C01811=1012.255,117.032,374.346,169.499,79.664,168.490
C01812=1012.256,116.639,374.386,169.507,79.676,168.501
C01813=1012.257,116.245,374.424,169.516,79.687,168.512
C01814=1012.259,115.850,374.464,169.527,79.699,168.525
C01815=1012.260,115.456,374.502,169.537,79.712,168.537
C01816=1012.261,115.062,374.541,169.547,79.725,168.549
C01817=1012.262,114.667,374.580,169.559,79.737,168.563
C01818=1012.263,114.273,374.619,169.567,79.748,168.573
C01819=1012.264,113.879,374.658,169.578,79.759,168.585
C01820=1012.266,113.484,374.697,169.586,79.770,168.596
C01821=1012.267,113.090,374.735,169.596,79.781,168.607
C01822=1012.269,112.696,374.774,169.607,79.793,168.620
C01823=1012.270,112.302,374.813,169.618,79.805,168.633
C01824=1012.271,111.908,374.852,169.629,79.818,168.646
C01825=1012.272,111.514,374.890,169.637,79.830,168.657
C01826=1012.273,111.119,374.929,169.651,79.841,168.671
C01827=1012.274,110.725,374.968,169.660,79.852,168.682
C01828=1012.275,110.331,375.007,169.670,79.863,168.694
C01829=1012.277,109.936,375.046,169.677,79.873,168.704
C01830=1012.278,109.542,375.084,169.689,79.885,168.717
C01831=1012.280,109.148,375.123,169.700,79.898,168.730
C01832=1012.280,108.754,375.162,169.709,79.909,168.741
C01833=1012.282,108.359,375.200,169.721,79.921,168.755
C01834=1012.283,107.965,375.239,169.730,79.932,168.766
C01835=1012.284,107.570,375.278,169.740,79.943,168.778
C01836=1012.285,107.176,375.316,169.751,79.954,168.790
C01837=1012.286,106.782,375.355,169.761,79.964,168.802
C01838=1012.287,106.388,375.394,169.771,79.976,168.814
C01839=1012.289,105.993,375.431,169.780,79.987,168.825
C01840=1012.290,105.599,375.470,169.792,79.999,168.839
C01841=1012.291,105.205,375.509,169.801,80.010,168.850
C01842=1012.292,104.811,375.547,169.815,80.022,168.865
C01843=1012.293,104.416,375.585,169.825,80.033,168.877
C01844=1012.295,104.022,375.624,169.832,80.043,168.886
C01845=1012.296,103.628,375.663,169.845,80.053,168.899
C01846=1012.296,103.233,375.702,169.852,80.063,168.909
C01847=1012.298,102.838,375.740,169.865,80.075,168.923
C01848=1012.299,102.444,375.778,169.877,80.087,168.937
C01849=1012.300,102.049,375.816,169.887,80.098,168.949
C01850=1012.301,101.655,375.855,169.898,80.109,168.962
C01851=1012.302,101.261,375.893,169.909,80.120,168.974
C01852=1012.304,100.866,375.932,169.920,80.130,168.987
C01853=1012.305,100.472,375.970,169.928,80.140,168.996
C01854=1012.307,100.077,376.008,169.937,80.149,169.007
C01855=1012.307,99.683,376.046,169.950,80.161,169.022
C01856=1012.309,99.288,376.085,169.960,80.173,169.033
C01857=1012.310,98.894,376.124,169.973,80.185,169.048
C01858=1012.311,98.499,376.161,169.984,80.196,169.061
C01859=1012.312,98.105,376.200,169.995,80.206,169.073
C01860=1012.313,97.710,376.238,170.003,80.216,169.083
C01861=1012.314,97.316,376.276,170.016,80.226,169.097
C01862=1012.316,96.921,376.314,170.025,80.235,169.108
C01863=1012.317,96.527,376.353,170.037,80.246,169.121
C01864=1012.318,96.133,376.391,170.047,80.257,169.133
C01865=1012.319,95.737,376.429,170.057,80.269,169.145
C01866=1012.320,95.343,376.467,170.068,80.279,169.158
C01867=1012.321,94.949,376.505,170.080,80.290,169.171
C01868=1012.322,94.554,376.543,170.089,80.299,169.182
C01869=1012.323,94.160,376.581,170.101,80.310,169.195
C01870=1012.325,93.765,376.619,170.111,80.319,169.206
C01871=1012.326,93.370,376.658,170.120,80.328,169.217
C01872=1012.327,92.976,376.696,170.132,80.339,169.230
C01873=1012.328,92.581,376.734,170.140,80.349,169.240
C01874=1012.329,92.186,376.772,170.152,80.360,169.253
C01875=1012.331,91.792,376.810,170.164,80.370,169.267
C01876=1012.332,91.397,376.847,170.176,80.381,169.280
C01877=1012.332,90.994,376.887,170.188,80.391,169.293
C01878=1012.333,90.749,376.911,170.195,80.397,169.301
C01879=1012.334,90.468,376.937,170.200,80.404,169.308
C01880=1012.335,90.194,376.963,170.207,80.410,169.316
C01881=1012.335,89.959,376.986,170.214,80.416,169.323
C01882=1012.336,89.564,377.024,170.224,80.426,169.334
C01883=1012.338,89.178,377.061,170.237,80.436,169.348
C01884=1012.339,88.800,377.097,170.246,80.445,169.359
C01885=1012.340,88.425,377.133,170.256,80.455,169.370
C01886=1012.341,88.047,377.170,170.266,80.464,169.382
C01887=1012.342,87.663,377.207,170.279,80.474,169.396
C01888=1012.343,87.269,377.244,170.288,80.484,169.407
C01889=1012.344,86.870,377.282,170.298,80.493,169.418
C01890=1012.345,86.469,377.320,170.311,80.504,169.432
C01891=1012.346,86.067,377.359,170.321,80.513,169.443
C01892=1012.347,85.664,377.398,170.333,80.524,169.457
C01893=1012.349,85.260,377.437,170.343,80.533,169.469
C01894=1012.350,84.853,377.476,170.356,80.543,169.482
C01895=1012.351,84.447,377.514,170.366,80.553,169.494
C01896=1012.352,84.039,377.554,170.378,80.563,169.508
C01897=1012.352,83.629,377.592,170.389,80.573,169.520
C01898=1012.354,83.218,377.632,170.401,80.583,169.533
C01899=1012.355,82.805,377.671,170.412,80.592,169.545
C01900=1012.356,82.393,377.710,170.424,80.603,169.559
C01901=1012.357,81.979,377.750,170.435,80.612,169.571
C01902=1012.358,81.565,377.789,170.447,80.623,169.585
C01903=1012.360,81.171,377.827,170.458,80.632,169.597
C01904=1012.360,80.807,377.862,170.470,80.641,169.609
C01905=1012.362,80.424,377.898,170.481,80.650,169.621
C01906=1012.363,80.012,377.936,170.490,80.660,169.633
C01907=1012.363,79.603,377.976,170.501,80.669,169.645
C01908=1012.364,79.201,378.014,170.511,80.678,169.657
C01909=1012.366,78.806,378.051,170.526,80.688,169.672
C01910=1012.366,78.417,378.088,170.536,80.698,169.684
C01911=1012.368,78.033,378.125,170.545,80.705,169.694
C01912=1012.368,77.652,378.161,170.556,80.715,169.706
C01913=1012.370,77.270,378.197,170.567,80.724,169.718
C01914=1012.371,76.884,378.234,170.578,80.733,169.730
C01915=1012.371,76.489,378.271,170.590,80.742,169.743
C01916=1012.372,76.088,378.309,170.601,80.751,169.755
C01917=1012.373,75.678,378.347,170.612,80.760,169.767
C01918=1012.374,75.264,378.387,170.623,80.769,169.780
C01919=1012.375,75.055,378.407,170.628,80.774,169.786
C01920=1012.376,74.840,378.427,170.636,80.780,169.794
C01921=1012.376,74.614,378.448,170.642,80.784,169.801
C01922=1012.377,74.385,378.470,170.647,80.789,169.807
C01923=1012.378,74.166,378.490,170.656,80.795,169.815
C01924=1012.379,73.752,378.530,170.667,80.804,169.828
C01925=1012.380,73.339,378.569,170.678,80.813,169.840
C01926=1012.381,72.930,378.607,170.689,80.823,169.853
C01927=1012.382,72.522,378.645,170.700,80.832,169.865
C01928=1012.383,72.116,378.683,170.711,80.841,169.878
C01929=1012.384,71.711,378.722,170.724,80.850,169.891
C01930=1012.384,71.306,378.760,170.735,80.859,169.903
C01931=1012.385,70.901,378.798,170.747,80.868,169.916
C01932=1012.386,70.497,378.836,170.756,80.876,169.926
C01933=1012.387,70.093,378.874,170.767,80.885,169.939
C01934=1012.388,69.689,378.912,170.779,80.894,169.952
C01935=1012.390,69.280,378.951,170.792,80.903,169.965
C01936=1012.391,68.864,378.989,170.803,80.912,169.978
C01937=1012.392,68.447,379.029,170.815,80.921,169.991
C01938=1012.393,68.035,379.067,170.824,80.929,170.001
C01939=1012.393,67.634,379.105,170.835,80.938,170.014
C01940=1012.395,67.235,379.142,170.848,80.947,170.027
C01941=1012.395,66.838,379.179,170.856,80.956,170.037
C01942=1012.396,66.474,379.213,170.867,80.963,170.049
C01943=1012.397,66.147,379.243,170.877,80.970,170.059
C01944=1012.398,65.754,379.281,170.886,80.978,170.070
C01945=1012.398,65.546,379.300,170.893,80.983,170.077
C01946=1012.399,65.331,379.320,170.899,80.987,170.084
C01947=1012.400,65.112,379.340,170.905,80.992,170.090
C01948=1012.400,64.890,379.361,170.911,80.996,170.097
C01949=1012.401,64.663,379.382,170.920,81.002,170.106
C01950=1012.401,64.436,379.403,170.926,81.006,170.113
C01951=1012.402,64.217,379.424,170.932,81.011,170.119
C01952=1012.402,63.813,379.460,170.977,81.046,170.169
C01953=1012.402,63.601,379.477,171.070,81.117,170.271
C01954=1012.402,63.366,379.495,171.175,81.195,170.386
C01955=1012.402,63.117,379.514,171.288,81.278,170.511
C01956=1012.402,62.875,379.533,171.401,81.358,170.633
C01957=1012.402,62.656,379.550,171.504,81.430,170.745
C01958=1012.402,62.372,379.572,171.641,81.524,170.894
C01959=1012.402,61.974,379.603,171.838,81.655,171.108
C01960=1012.402,61.578,379.633,172.039,81.784,171.326
C01961=1012.403,61.182,379.664,172.249,81.914,171.552
C01962=1012.402,60.785,379.695,172.466,82.043,171.786
C01963=1012.403,60.389,379.726,172.690,82.171,172.025
C01964=1012.403,59.993,379.756,172.921,82.299,172.272
C01965=1012.402,59.598,379.787,173.157,82.427,172.524
C01966=1012.403,59.201,379.818,173.408,82.554,172.791
C01967=1012.403,58.805,379.848,173.660,82.680,173.059
C01968=1012.403,58.409,379.880,173.927,82.807,173.341
C01969=1012.403,58.013,379.910,174.202,82.932,173.630
C01970=1012.403,57.616,379.940,174.486,83.058,173.930
C01971=1012.403,57.221,379.972,174.784,83.183,174.242
C01972=1012.403,56.824,380.002,175.090,83.306,174.562
C01973=1012.404,56.429,380.033,175.408,83.430,174.895
C01974=1012.404,56.033,380.063,175.735,83.552,175.237
C01975=1012.404,55.636,380.094,176.082,83.675,175.597
C01976=1012.404,55.241,380.125,176.433,83.797,175.963
C01977=1012.404,54.844,380.155,176.806,83.918,176.349
C01978=1012.405,54.448,380.186,177.189,84.039,176.746
C01979=1012.404,54.052,380.217,177.590,84.158,177.160
C01980=1012.405,53.656,380.247,178.004,84.277,177.588
C01981=1012.405,53.260,380.278,178.436,84.396,178.033
C01982=1012.406,52.865,380.309,178.889,84.513,178.499
C01983=1012.406,52.469,380.339,179.364,84.631,178.987
C01984=1012.407,52.072,380.370,179.855,84.746,179.490
C01985=1012.407,51.677,380.400,-179.631,84.863,-179.983
C01986=1012.407,51.281,380.431,-179.099,84.977,-179.438
C01987=1012.407,50.884,380.461,-178.540,85.091,-178.867
C01988=1012.407,50.489,380.492,-177.953,85.203,-178.268
C01989=1012.408,50.093,380.522,-177.344,85.315,-177.647
C01990=1012.408,49.697,380.553,-176.695,85.427,-176.986
C01991=1012.409,49.301,380.584,-176.030,85.537,-176.309
C01992=1012.409,48.905,380.614,-175.320,85.647,-175.588
C01993=1012.410,48.508,380.645,-174.582,85.754,-174.838
C01994=1012.410,48.114,380.675,-173.803,85.862,-174.048
C01995=1012.411,47.717,380.706,-172.982,85.967,-173.216
C01996=1012.411,47.321,380.736,-172.125,86.072,-172.348
C01997=1012.412,46.926,380.767,-171.221,86.176,-171.432
C01998=1012.412,46.530,380.798,-170.277,86.277,-170.478
C01999=1012.411,46.134,380.828,-169.265,86.378,-169.456
C02000=1012.413,45.739,380.859,-168.208,86.477,-168.388
C02001=1012.413,45.342,380.889,-167.101,86.574,-167.271
C02002=1012.413,44.947,380.920,-165.914,86.670,-166.074
C02003=1012.414,44.551,380.950,-164.672,86.764,-164.822
C02004=1012.414,44.155,380.982,-163.370,86.855,-163.509
C02005=1012.415,43.760,381.011,-161.972,86.945,-162.102
C02006=1012.415,43.364,381.042,-160.504,87.033,-160.624
C02007=1012.416,42.969,381.073,-158.950,87.118,-159.060
C02008=1012.416,42.572,381.103,-157.318,87.201,-157.418
C02009=1012.417,42.177,381.134,-155.591,87.280,-155.683
C02010=1012.417,41.781,381.165,-153.754,87.358,-153.836
C02011=1012.418,41.386,381.194,-151.813,87.432,-151.886
C02012=1012.418,40.990,381.225,-149.777,87.502,-149.842
C02013=1012.419,40.594,381.256,-147.632,87.569,-147.689
C02014=1012.419,40.200,381.286,-145.391,87.631,-145.438
C02015=1012.420,39.803,381.317,-143.005,87.690,-143.044
C02016=1012.420,39.408,381.347,-140.520,87.745,-140.550
C02017=1012.421,39.012,381.378,-137.951,87.794,-137.973
C02018=1012.422,38.616,381.408,-135.243,87.839,-135.257
C02019=1012.423,38.221,381.439,-132.449,87.879,-132.455
C02020=1012.423,37.825,381.469,-129.568,87.913,-129.567
C02021=1012.423,37.430,381.499,-126.623,87.942,-126.613
C02022=1012.424,37.035,381.530,-123.575,87.965,-123.558
C02023=1012.424,36.639,381.561,-120.534,87.982,-120.509
C02024=1012.425,36.243,381.591,-117.404,87.993,-117.372
C02025=1012.426,35.849,381.622,-114.310,87.998,-114.271
C02026=1012.427,35.453,381.652,-111.189,87.997,-111.142
C02027=1012.427,35.057,381.682,-108.098,87.990,-108.044
C02028=1012.428,34.662,381.713,-105.036,87.977,-104.976
C02029=1012.429,34.266,381.743,-102.042,87.959,-101.975
C02030=1012.430,33.871,381.774,-99.149,87.936,-99.074
C02031=1012.430,33.475,381.804,-96.307,87.906,-96.226
C02032=1012.430,33.080,381.835,-93.566,87.873,-93.479
C02033=1012.431,32.685,381.865,-90.937,87.834,-90.843
C02034=1012.432,32.290,381.896,-88.403,87.792,-88.303
C02035=1012.433,31.894,381.926,-85.985,87.745,-85.878
C02036=1012.433,31.499,381.957,-83.686,87.695,-83.574
C02037=1012.434,31.103,381.987,-81.471,87.641,-81.352
C02038=1012.434,30.708,382.018,-79.404,87.585,-79.280
C02039=1012.435,30.313,382.047,-77.406,87.524,-77.277
C02040=1012.436,29.917,382.078,-75.542,87.463,-75.406
C02041=1012.436,29.522,382.108,-73.759,87.398,-73.618
C02042=1012.437,29.127,382.139,-72.088,87.331,-71.941
C02043=1012.438,28.732,382.169,-70.499,87.263,-70.348
C02044=1012.439,28.338,382.200,-68.990,87.192,-68.833
C02045=1012.439,27.944,382.230,-67.576,87.120,-67.414
C02046=1012.440,27.552,382.260,-66.231,87.047,-66.065
C02047=1012.441,27.158,382.291,-64.958,86.973,-64.786
C02048=1012.441,26.764,382.321,-63.759,86.898,-63.582
C02049=1012.442,26.368,382.352,-62.613,86.821,-62.432
C02050=1012.443,25.970,382.383,-61.514,86.743,-61.328
C02051=1012.443,25.570,382.413,-60.479,86.664,-60.288
C02052=1012.444,25.174,382.443,-59.503,86.584,-59.308
C02053=1012.445,24.779,382.474,-58.575,86.504,-58.376
C02054=1012.446,24.383,382.504,-57.689,86.424,-57.485
C02055=1012.447,24.004,382.534,-56.888,86.347,-56.681
C02056=1012.447,23.664,382.560,-56.198,86.277,-55.987
C02057=1012.448,23.248,382.591,-55.397,86.192,-55.182
C02058=1012.448,22.884,382.620,-54.721,86.116,-54.503
C02059=1012.449,22.606,382.641,-54.231,86.059,-54.009
C02060=1012.450,22.275,382.667,-53.666,85.990,-53.442
C02061=1012.450,21.947,382.692,-53.123,85.921,-52.895
C02062=1012.451,21.558,382.721,-52.509,85.841,-52.278
C02063=1012.451,21.330,382.740,-52.158,85.793,-51.925
C02064=1012.452,21.083,382.759,-51.791,85.742,-51.556
C02065=1012.452,20.822,382.778,-51.416,85.687,-51.178
C02066=1012.453,20.554,382.799,-51.042,85.631,-50.802
C02067=1012.454,20.285,382.819,-50.678,85.576,-50.436
C02068=1012.454,20.024,382.840,-50.331,85.521,-50.087
C02069=1012.455,19.782,382.858,-50.022,85.471,-49.776
C02070=1012.455,19.561,382.875,-49.742,85.424,-49.494
C02071=1012.456,19.358,382.891,-49.496,85.383,-49.247
C02072=1012.456,18.955,382.922,-49.018,85.299,-48.766
C02073=1012.457,18.555,382.952,-48.564,85.216,-48.309
C02074=1012.457,18.163,382.983,-48.132,85.135,-47.873
C02075=1012.458,17.773,383.013,-47.720,85.053,-47.459
C02076=1012.460,17.386,383.043,-47.329,84.973,-47.065
C02077=1012.460,16.999,383.073,-46.955,84.894,-46.689
C02078=1012.460,16.615,383.102,-46.594,84.815,-46.325
C02079=1012.461,16.232,383.131,-46.249,84.737,-45.978
C02080=1012.462,15.851,383.161,-45.914,84.658,-45.641
C02081=1012.463,15.471,383.190,-45.594,84.581,-45.319
C02082=1012.464,15.090,383.220,-45.284,84.503,-45.006
C02083=1012.464,14.710,383.249,-44.988,84.426,-44.709
C02084=1012.465,14.330,383.278,-44.699,84.350,-44.418
C02085=1012.466,13.949,383.307,-44.419,84.273,-44.136
C02086=1012.467,13.567,383.337,-44.146,84.196,-43.861
C02087=1012.468,13.184,383.366,-43.885,84.121,-43.598
C02088=1012.468,12.800,383.396,-43.626,84.044,-43.337
C02089=1012.468,12.416,383.425,-43.379,83.967,-43.089
C02090=1012.470,12.034,383.454,-43.142,83.892,-42.851
C02091=1012.470,11.662,383.483,-42.919,83.820,-42.626
C02092=1012.471,11.298,383.511,-42.705,83.749,-42.409
C02093=1012.472,10.933,383.540,-42.496,83.677,-42.200
C02094=1012.472,10.559,383.568,-42.292,83.605,-41.995
C02095=1012.473,10.181,383.598,-42.089,83.533,-41.790
C02096=1012.474,9.805,383.626,-41.894,83.461,-41.594
C02097=1012.475,9.431,383.655,-41.703,83.390,-41.401
C02098=1012.475,9.057,383.684,-41.520,83.319,-41.218
C02099=1012.475,8.683,383.713,-41.342,83.248,-41.038
C02100=1012.477,8.309,383.741,-41.166,83.178,-40.861
C02101=1012.478,7.933,383.771,-40.998,83.108,-40.692
C02102=1012.478,7.555,383.799,-40.833,83.039,-40.527
C02103=1012.479,7.173,383.828,-40.668,82.968,-40.361
C02104=1012.480,6.788,383.858,-40.512,82.898,-40.204
C02105=1012.480,6.396,383.888,-40.353,82.827,-40.045
C02106=1012.482,6.004,383.919,-40.199,82.755,-39.890
C02107=1012.481,5.611,383.949,-40.051,82.685,-39.742
C02108=1012.483,5.220,383.979,-39.906,82.615,-39.596
C02109=1012.483,4.832,384.009,-39.766,82.546,-39.455
C02110=1012.485,4.442,384.039,-39.628,82.478,-39.317
C02111=1012.485,4.051,384.070,-39.493,82.410,-39.180
C02112=1012.486,3.679,384.098,-39.371,82.345,-39.060
C02113=1012.487,3.335,384.125,-39.259,82.285,-38.947
C02114=1012.487,3.010,384.149,-39.155,82.230,-38.843
C02115=1012.487,2.687,384.174,-39.056,82.175,-38.743
C02116=1012.489,2.345,384.201,-38.951,82.117,-38.638
C02117=1012.488,1.974,384.229,-38.840,82.055,-38.527
C02118=1012.490,1.582,384.260,-38.727,81.989,-38.414
C02119=1012.490,1.185,384.290,-38.616,81.924,-38.303
C02120=1012.491,0.788,384.321,-38.507,81.858,-38.194
C02121=1012.492,0.394,384.351,-38.402,81.794,-38.089
C02122=1012.492,-0.001,384.381,-38.298,81.730,-37.985
C02123=1012.493,-0.399,384.412,-38.196,81.666,-37.883
C02124=1012.494,-0.800,384.443,-38.099,81.602,-37.787
C02125=1012.494,-1.202,384.474,-37.999,81.539,-37.686
C02126=1012.496,-1.606,384.505,-37.905,81.475,-37.593
C02127=1012.496,-2.013,384.536,-37.811,81.413,-37.499
C02128=1012.497,-2.422,384.568,-37.719,81.350,-37.407
C02129=1012.497,-2.832,384.599,-37.630,81.288,-37.319
C02130=1012.498,-3.244,384.631,-37.543,81.226,-37.233
C02131=1012.498,-3.645,384.662,-37.458,81.166,-37.148
C02132=1012.499,-4.031,384.691,-37.381,81.109,-37.071
C02133=1012.500,-4.410,384.721,-37.307,81.053,-36.998
C02134=1012.501,-4.801,384.751,-37.229,80.996,-36.920
C02135=1012.501,-5.215,384.783,-37.151,80.937,-36.843
C02136=1012.502,-5.430,384.800,-37.110,80.906,-36.802
C02137=1012.501,-5.646,384.816,-37.074,80.875,-36.767
C02138=1012.502,-5.863,384.833,-37.034,80.844,-36.727
C02139=1012.503,-6.080,384.850,-36.994,80.813,-36.687
C02140=1012.503,-6.296,384.866,-36.957,80.783,-36.651
C02141=1012.504,-6.513,384.883,-36.919,80.754,-36.613
C02142=1012.504,-6.729,384.899,-36.883,80.724,-36.578
C02143=1012.505,-6.945,384.917,-36.845,80.695,-36.540
C02144=1012.505,-7.159,384.933,-36.809,80.664,-36.505
C02145=1012.504,-7.374,384.949,-36.775,80.636,-36.471
C02146=1012.506,-7.587,384.966,-36.739,80.607,-36.435
C02147=1012.505,-7.800,384.983,-36.705,80.578,-36.401
C02148=1012.506,-8.013,384.999,-36.671,80.549,-36.368
C02149=1012.506,-8.224,385.015,-36.639,80.522,-36.337
C02150=1012.506,-8.436,385.032,-36.606,80.494,-36.304
C02151=1012.506,-8.647,385.048,-36.574,80.467,-36.273
C02152=1012.507,-8.858,385.064,-36.541,80.438,-36.241
C02153=1012.508,-9.070,385.081,-36.510,80.411,-36.210
C02154=1012.508,-9.281,385.097,-36.479,80.384,-36.179
C02155=1012.508,-9.703,385.129,-36.419,80.330,-36.121
C02156=1012.509,-10.124,385.162,-36.360,80.278,-36.062
C02157=1012.509,-10.544,385.194,-36.302,80.224,-36.006
C02158=1012.511,-10.963,385.226,-36.245,80.173,-35.949
C02159=1012.511,-11.381,385.259,-36.191,80.123,-35.896
C02160=1012.512,-11.797,385.291,-36.137,80.072,-35.843
C02161=1012.512,-12.212,385.322,-36.085,80.024,-35.792
C02162=1012.513,-12.625,385.354,-36.036,79.975,-35.745
C02163=1012.514,-13.034,385.386,-35.986,79.928,-35.696
C02164=1012.514,-13.433,385.417,-35.941,79.883,-35.651
C02165=1012.514,-13.820,385.446,-35.897,79.839,-35.610
C02166=1012.515,-14.197,385.476,-35.857,79.797,-35.570
C02167=1012.516,-14.572,385.504,-35.816,79.756,-35.531
C02168=1012.516,-14.948,385.534,-35.775,79.716,-35.491
C02169=1012.517,-15.332,385.563,-35.738,79.675,-35.455
C02170=1012.517,-15.723,385.594,-35.699,79.634,-35.418
C02171=1012.518,-16.120,385.625,-35.659,79.594,-35.378
C02172=1012.518,-16.515,385.655,-35.622,79.553,-35.344
C02173=1012.519,-16.914,385.686,-35.585,79.513,-35.308
C02174=1012.520,-17.309,385.716,-35.547,79.474,-35.270
C02175=1012.520,-17.695,385.746,-35.514,79.437,-35.238
C02176=1012.521,-17.899,385.761,-35.497,79.417,-35.222
C02177=1012.521,-18.124,385.779,-35.476,79.396,-35.202
C02178=1012.521,-18.377,385.798,-35.456,79.371,-35.184
C02179=1012.521,-18.650,385.820,-35.434,79.346,-35.163
C02180=1012.521,-18.929,385.841,-35.411,79.321,-35.140
C02181=1012.522,-19.204,385.862,-35.389,79.295,-35.119
C02182=1012.522,-19.460,385.882,-35.368,79.272,-35.099
C02183=1012.522,-19.691,385.900,-35.350,79.252,-35.081
C02184=1012.522,-19.896,385.916,-35.334,79.234,-35.066
C02185=1012.523,-20.246,385.943,-35.308,79.203,-35.041
C02186=1012.524,-20.643,385.974,-35.280,79.170,-35.015
C02187=1012.524,-21.036,386.004,-35.251,79.137,-34.987
C02188=1012.524,-21.430,386.034,-35.225,79.105,-34.962
C02189=1012.524,-21.823,386.064,-35.198,79.073,-34.937
C02190=1012.525,-22.216,386.095,-35.172,79.041,-34.913
C02191=1012.526,-22.609,386.126,-35.149,79.011,-34.891
C02192=1012.526,-23.002,386.156,-35.123,78.981,-34.866
C02193=1012.526,-23.396,386.187,-35.100,78.951,-34.845
C02194=1012.527,-23.790,386.216,-35.078,78.923,-34.824
C02195=1012.527,-24.183,386.247,-35.055,78.896,-34.802
C02196=1012.528,-24.576,386.277,-35.034,78.867,-34.783
C02197=1012.528,-24.969,386.308,-35.013,78.841,-34.763
C02198=1012.528,-25.362,386.338,-34.991,78.815,-34.742
C02199=1012.529,-25.756,386.369,-34.973,78.789,-34.726
C02200=1012.529,-26.149,386.398,-34.953,78.764,-34.707
C02201=1012.529,-26.543,386.429,-34.935,78.740,-34.690
C02202=1012.530,-26.936,386.460,-34.919,78.717,-34.677
C02203=1012.530,-27.329,386.490,-34.901,78.693,-34.659
C02204=1012.530,-27.723,386.521,-34.885,78.672,-34.645
C02205=1012.531,-28.117,386.551,-34.869,78.649,-34.630
C02206=1012.531,-28.510,386.582,-34.852,78.629,-34.614
C02207=1012.531,-28.903,386.612,-34.838,78.608,-34.602
C02208=1012.532,-29.297,386.643,-34.824,78.588,-34.589
C02209=1012.531,-29.690,386.673,-34.811,78.570,-34.578
C02210=1012.532,-30.084,386.703,-34.799,78.551,-34.567
C02211=1012.533,-30.477,386.734,-34.787,78.533,-34.556
C02212=1012.533,-30.870,386.764,-34.775,78.516,-34.546
C02213=1012.533,-31.264,386.795,-34.762,78.499,-34.534
C02214=1012.533,-31.658,386.824,-34.752,78.484,-34.524
C02215=1012.534,-32.051,386.855,-34.742,78.469,-34.517
C02216=1012.534,-32.444,386.885,-34.732,78.454,-34.508
C02217=1012.534,-32.838,386.916,-34.724,78.441,-34.501
C02218=1012.534,-33.232,386.947,-34.716,78.427,-34.495
C02219=1012.535,-33.626,386.977,-34.708,78.414,-34.488
C02220=1012.534,-34.019,387.007,-34.701,78.402,-34.482
C02221=1012.535,-34.412,387.038,-34.694,78.392,-34.476
C02222=1012.535,-34.805,387.068,-34.689,78.381,-34.473
C02223=1012.535,-35.199,387.099,-34.682,78.370,-34.467
C02224=1012.535,-35.592,387.129,-34.676,78.362,-34.462
C02225=1012.536,-35.986,387.160,-34.671,78.353,-34.457
C02226=1012.536,-36.379,387.190,-34.667,78.345,-34.455
C02227=1012.536,-36.773,387.221,-34.665,78.338,-34.454
C02228=1012.536,-37.166,387.251,-34.661,78.331,-34.452
C02229=1012.536,-37.560,387.282,-34.658,78.325,-34.450
C02230=1012.536,-37.953,387.312,-34.656,78.320,-34.449
C02231=1012.537,-38.346,387.343,-34.655,78.316,-34.449
C02232=1012.537,-38.740,387.373,-34.653,78.311,-34.448
C02233=1012.536,-39.133,387.404,-34.654,78.308,-34.451
C02234=1012.537,-39.527,387.434,-34.654,78.305,-34.452
C02235=1012.537,-39.920,387.464,-34.654,78.304,-34.452
C02236=1012.538,-40.313,387.495,-34.656,78.302,-34.456
C02237=1012.538,-40.707,387.525,-34.656,78.302,-34.456
C02238=1012.537,-41.100,387.555,-34.658,78.301,-34.460
C02239=1012.538,-41.493,387.586,-34.662,78.303,-34.464
C02240=1012.538,-41.886,387.617,-34.665,78.304,-34.469
C02241=1012.537,-42.279,387.647,-34.669,78.306,-34.474
C02242=1012.538,-42.672,387.678,-34.673,78.309,-34.479
C02243=1012.538,-43.065,387.708,-34.677,78.312,-34.484
C02244=1012.538,-43.459,387.739,-34.682,78.316,-34.490
C02245=1012.537,-43.852,387.769,-34.689,78.321,-34.498
C02246=1012.538,-44.245,387.800,-34.694,78.326,-34.504
C02247=1012.538,-44.638,387.830,-34.702,78.333,-34.512
C02248=1012.537,-45.031,387.861,-34.710,78.340,-34.521
C02249=1012.538,-45.423,387.891,-34.717,78.347,-34.530
C02250=1012.538,-45.816,387.921,-34.726,78.355,-34.539
C02251=1012.538,-46.210,387.952,-34.734,78.363,-34.548
C02252=1012.538,-46.602,387.983,-34.744,78.374,-34.558
C02253=1012.538,-46.995,388.013,-34.755,78.384,-34.570
C02254=1012.538,-47.388,388.043,-34.764,78.394,-34.580
C02255=1012.538,-47.780,388.074,-34.776,78.407,-34.593
C02256=1012.537,-48.173,388.104,-34.788,78.419,-34.605
C02257=1012.538,-48.565,388.135,-34.800,78.431,-34.618
C02258=1012.537,-48.958,388.165,-34.813,78.445,-34.632
C02259=1012.537,-49.352,388.195,-34.826,78.459,-34.645
C02260=1012.537,-49.743,388.226,-34.840,78.474,-34.661
C02261=1012.537,-50.136,388.256,-34.856,78.490,-34.677
C02262=1012.537,-50.529,388.287,-34.871,78.506,-34.694
C02263=1012.537,-50.922,388.317,-34.886,78.523,-34.708
C02264=1012.537,-51.314,388.348,-34.903,78.541,-34.726
C02265=1012.537,-51.707,388.379,-34.921,78.560,-34.745
C02266=1012.537,-52.100,388.410,-34.937,78.578,-34.761
C02267=1012.537,-52.492,388.440,-34.956,78.599,-34.781
C02268=1012.537,-52.885,388.470,-34.976,78.619,-34.802
C02269=1012.536,-53.278,388.500,-34.994,78.640,-34.820
C02270=1012.536,-53.669,388.531,-35.015,78.661,-34.842
C02271=1012.536,-54.063,388.561,-35.036,78.685,-34.863
C02272=1012.536,-54.454,388.592,-35.058,78.708,-34.885
C02273=1012.536,-54.847,388.622,-35.079,78.731,-34.908
C02274=1012.535,-55.240,388.653,-35.102,78.756,-34.930
C02275=1012.536,-55.632,388.683,-35.127,78.781,-34.956
C02276=1012.535,-56.025,388.714,-35.151,78.807,-34.981
C02277=1012.535,-56.418,388.744,-35.175,78.833,-35.005
C02278=1012.535,-56.811,388.774,-35.201,78.861,-35.032
C02279=1012.535,-57.205,388.805,-35.228,78.889,-35.059
C02280=1012.535,-57.598,388.836,-35.255,78.918,-35.087
C02281=1012.535,-57.993,388.867,-35.282,78.947,-35.114
C02282=1012.534,-58.388,388.897,-35.311,78.977,-35.143
C02283=1012.534,-58.783,388.928,-35.341,79.008,-35.174
C02284=1012.534,-59.178,388.958,-35.371,79.040,-35.203
C02285=1012.534,-59.575,388.990,-35.403,79.072,-35.236
C02286=1012.533,-59.972,389.020,-35.436,79.106,-35.269
C02287=1012.533,-60.369,389.051,-35.468,79.139,-35.302
C02288=1012.533,-60.767,389.083,-35.502,79.175,-35.336
C02289=1012.533,-61.166,389.113,-35.538,79.209,-35.373
C02290=1012.533,-61.564,389.144,-35.572,79.246,-35.406
C02291=1012.532,-61.964,389.174,-35.611,79.283,-35.446
C02292=1012.532,-62.363,389.206,-35.647,79.320,-35.482
C02293=1012.532,-62.764,389.238,-35.686,79.358,-35.522
C02294=1012.531,-63.165,389.268,-35.726,79.398,-35.562
C02295=1012.532,-63.567,389.300,-35.769,79.438,-35.605
C02296=1012.531,-63.968,389.331,-35.811,79.479,-35.647
C02297=1012.531,-64.370,389.362,-35.853,79.520,-35.689
C02298=1012.530,-64.772,389.393,-35.897,79.562,-35.733
C02299=1012.530,-65.175,389.425,-35.941,79.605,-35.777
C02300=1012.530,-65.578,389.456,-35.989,79.649,-35.826
C02301=1012.529,-65.981,389.487,-36.035,79.693,-35.872
C02302=1012.529,-66.385,389.519,-36.084,79.738,-35.921
C02303=1012.529,-66.789,389.550,-36.135,79.783,-35.973
C02304=1012.528,-67.192,389.582,-36.188,79.830,-36.026
C02305=1012.528,-67.596,389.613,-36.238,79.878,-36.076
C02306=1012.527,-68.001,389.645,-36.293,79.926,-36.131
C02307=1012.527,-68.404,389.676,-36.349,79.975,-36.188
C02308=1012.527,-68.810,389.707,-36.404,80.024,-36.243
C02309=1012.527,-69.214,389.739,-36.463,80.074,-36.301
C02310=1012.526,-69.618,389.770,-36.524,80.125,-36.363
C02311=1012.526,-70.022,389.802,-36.584,80.177,-36.424
C02312=1012.526,-70.427,389.833,-36.645,80.229,-36.483
C02313=1012.525,-70.831,389.864,-36.709,80.281,-36.549
C02314=1012.525,-71.235,389.896,-36.775,80.336,-36.614
C02315=1012.525,-71.639,389.927,-36.842,80.390,-36.682
C02316=1012.524,-72.043,389.959,-36.912,80.445,-36.752
C02317=1012.524,-72.447,389.990,-36.982,80.501,-36.823
C02318=1012.523,-72.851,390.022,-37.055,80.557,-36.896
C02319=1012.523,-73.255,390.054,-37.128,80.615,-36.968
C02320=1012.523,-73.659,390.085,-37.205,80.673,-37.046
C02321=1012.522,-74.061,390.116,-37.282,80.731,-37.123
C02322=1012.522,-74.465,390.147,-37.362,80.791,-37.203
C02323=1012.522,-74.868,390.179,-37.444,80.850,-37.285
C02324=1012.521,-75.271,390.210,-37.527,80.911,-37.369
C02325=1012.521,-75.674,390.241,-37.613,80.971,-37.455
C02326=1012.521,-76.076,390.273,-37.702,81.033,-37.544
C02327=1012.520,-76.479,390.304,-37.791,81.096,-37.633
C02328=1012.519,-76.881,390.335,-37.884,81.160,-37.726
C02329=1012.520,-77.283,390.367,-37.978,81.223,-37.821
C02330=1012.519,-77.685,390.398,-38.076,81.288,-37.919
C02331=1012.518,-78.087,390.429,-38.175,81.353,-38.018
C02332=1012.518,-78.488,390.461,-38.279,81.418,-38.123
C02333=1012.518,-78.889,390.492,-38.383,81.485,-38.227
C02334=1012.517,-79.289,390.522,-38.492,81.552,-38.337
C02335=1012.517,-79.689,390.554,-38.602,81.619,-38.447
C02336=1012.516,-80.089,390.585,-38.714,81.686,-38.560
C02337=1012.516,-80.487,390.616,-38.830,81.756,-38.676
C02338=1012.516,-80.885,390.647,-38.952,81.824,-38.799
C02339=1012.515,-81.282,390.678,-39.072,81.894,-38.919
C02340=1012.515,-81.679,390.709,-39.196,81.964,-39.043
C02341=1012.515,-82.078,390.740,-39.325,82.035,-39.173
C02342=1012.514,-82.477,390.771,-39.461,82.107,-39.309
C02343=1012.514,-82.872,390.802,-39.595,82.178,-39.445
C02344=1012.513,-83.269,390.832,-39.735,82.251,-39.585
C02345=1012.513,-83.665,390.863,-39.881,82.324,-39.732
C02346=1012.513,-84.056,390.894,-40.025,82.397,-39.876
C02347=1012.512,-84.449,390.924,-40.177,82.470,-40.029
C02348=1012.512,-84.866,390.957,-40.342,82.549,-40.194
C02349=1012.512,-85.097,390.975,-40.437,82.594,-40.291
C02350=1012.511,-85.335,390.994,-40.533,82.639,-40.386
C02351=1012.511,-85.574,391.012,-40.637,82.685,-40.492
C02352=1012.511,-85.809,391.030,-40.736,82.730,-40.590
C02353=1012.511,-86.032,391.048,-40.833,82.774,-40.688
C02354=1012.510,-86.439,391.080,-41.017,82.853,-40.873
C02355=1012.510,-86.827,391.109,-41.194,82.929,-41.051
C02356=1012.510,-87.203,391.139,-41.373,83.004,-41.230
C02357=1012.509,-87.572,391.167,-41.552,83.077,-41.411
C02358=1012.509,-87.934,391.195,-41.736,83.150,-41.595
C02359=1012.508,-88.311,391.225,-41.930,83.226,-41.790
C02360=1012.508,-88.696,391.255,-42.136,83.304,-41.997
C02361=1012.508,-88.915,391.273,-42.255,83.349,-42.116
C02362=1012.508,-89.157,391.291,-42.389,83.399,-42.251
C02363=1012.508,-89.413,391.311,-42.538,83.451,-42.401
C02364=1012.507,-89.672,391.331,-42.688,83.504,-42.552
C02365=1012.507,-89.923,391.351,-42.837,83.557,-42.701
C02366=1012.507,-90.157,391.369,-42.981,83.606,-42.847
C02367=1012.506,-90.367,391.385,-43.112,83.650,-42.978
C02368=1012.506,-90.636,391.406,-43.280,83.706,-43.146
C02369=1012.506,-90.990,391.434,-43.511,83.781,-43.379
C02370=1012.506,-91.380,391.464,-43.774,83.863,-43.644
C02371=1012.505,-91.768,391.494,-44.044,83.946,-43.914
C02372=1012.505,-92.156,391.525,-44.321,84.029,-44.193
C02373=1012.505,-92.544,391.555,-44.610,84.113,-44.484
C02374=1012.505,-92.931,391.585,-44.909,84.197,-44.783
C02375=1012.504,-93.317,391.615,-45.221,84.281,-45.098
C02376=1012.504,-93.702,391.644,-45.538,84.365,-45.416
C02377=1012.504,-94.085,391.675,-45.870,84.449,-45.749
C02378=1012.503,-94.468,391.704,-46.217,84.533,-46.099
C02379=1012.502,-94.850,391.734,-46.571,84.619,-46.453
C02380=1012.503,-95.230,391.764,-46.941,84.703,-46.826
C02381=1012.503,-95.609,391.793,-47.318,84.787,-47.204
C02382=1012.503,-95.987,391.823,-47.713,84.872,-47.601
C02383=1012.502,-96.365,391.852,-48.129,84.957,-48.019
C02384=1012.501,-96.741,391.882,-48.552,85.041,-48.444
C02385=1012.501,-97.118,391.911,-48.997,85.126,-48.891
C02386=1012.501,-97.493,391.940,-49.458,85.211,-49.354
C02387=1012.501,-97.869,391.969,-49.943,85.297,-49.841
C02388=1012.501,-98.245,391.998,-50.447,85.381,-50.347
C02389=1012.500,-98.620,392.028,-50.970,85.467,-50.872
C02390=1012.500,-98.996,392.057,-51.521,85.553,-51.425
C02391=1012.500,-99.373,392.086,-52.102,85.639,-52.009
C02392=1012.500,-99.751,392.115,-52.699,85.724,-52.608
C02393=1012.499,-100.129,392.145,-53.338,85.811,-53.250
C02394=1012.499,-100.509,392.174,-54.004,85.897,-53.919
C02395=1012.499,-100.890,392.204,-54.710,85.984,-54.627
C02396=1012.499,-101.272,392.234,-55.448,86.071,-55.368
C02397=1012.499,-101.654,392.263,-56.229,86.157,-56.152
C02398=1012.499,-102.037,392.293,-57.049,86.244,-56.974
C02399=1012.498,-102.422,392.323,-57.918,86.330,-57.846
C02400=1012.498,-102.807,392.353,-58.841,86.417,-58.772
C02401=1012.498,-103.193,392.383,-59.811,86.502,-59.745
C02402=1012.498,-103.580,392.413,-60.840,86.587,-60.777
C02403=1012.498,-103.967,392.443,-61.925,86.672,-61.866
C02404=1012.498,-104.355,392.473,-63.071,86.756,-63.015
C02405=1012.497,-104.742,392.503,-64.290,86.839,-64.237
C02406=1012.497,-105.131,392.534,-65.593,86.922,-65.543
C02407=1012.497,-105.519,392.563,-66.967,87.002,-66.921
C02408=1012.497,-105.908,392.594,-68.416,87.081,-68.374
C02409=1012.496,-106.299,392.625,-69.981,87.160,-69.943
C02410=1012.496,-106.706,392.656,-71.709,87.240,-71.674
C02411=1012.497,-106.920,392.672,-72.649,87.280,-72.617
C02412=1012.497,-107.141,392.690,-73.666,87.322,-73.635
C02413=1012.497,-107.367,392.707,-74.739,87.364,-74.711
C02414=1012.497,-107.597,392.725,-75.872,87.405,-75.846
C02415=1012.496,-107.830,392.743,-77.059,87.446,-77.035
C02416=1012.497,-108.061,392.761,-78.283,87.486,-78.262
C02417=1012.497,-108.291,392.779,-79.529,87.525,-79.511
C02418=1012.496,-108.516,392.796,-80.802,87.561,-80.786
C02419=1012.497,-108.735,392.813,-82.077,87.596,-82.063
C02420=1012.497,-109.152,392.846,-84.628,87.659,-84.619
C02421=1012.496,-109.547,392.876,-87.159,87.713,-87.154
C02422=1012.496,-109.935,392.907,-89.789,87.763,-89.788
C02423=1012.496,-110.325,392.937,-92.552,87.808,-92.556
C02424=1012.496,-110.713,392.967,-95.443,87.848,-95.452
C02425=1012.496,-111.101,392.997,-98.432,87.882,-98.445
C02426=1012.496,-111.491,393.027,-101.550,87.911,-101.568
C02427=1012.496,-111.879,393.057,-104.764,87.933,-104.787
C02428=1012.497,-112.268,393.087,-108.034,87.948,-108.063
C02429=1012.497,-112.657,393.118,-111.365,87.957,-111.399
C02430=1012.496,-113.045,393.147,-114.711,87.959,-114.750
C02431=1012.497,-113.434,393.177,-118.069,87.953,-118.113
C02432=1012.497,-113.822,393.208,-121.419,87.941,-121.468
C02433=1012.497,-114.211,393.238,-124.757,87.921,-124.812
C02434=1012.497,-114.599,393.267,-127.995,87.894,-128.056
C02435=1012.497,-114.988,393.298,-131.188,87.861,-131.254
C02436=1012.498,-115.376,393.328,-134.262,87.821,-134.334
C02437=1012.497,-115.765,393.358,-137.236,87.775,-137.315
C02438=1012.498,-116.154,393.388,-140.115,87.722,-140.199
C02439=1012.498,-116.542,393.419,-142.853,87.663,-142.944
C02440=1012.498,-116.930,393.449,-145.450,87.600,-145.547
C02441=1012.499,-117.319,393.478,-147.927,87.532,-148.030
C02442=1012.499,-117.708,393.509,-150.291,87.458,-150.401
C02443=1012.499,-118.095,393.539,-152.504,87.380,-152.621
C02444=1012.499,-118.483,393.569,-154.595,87.299,-154.718
C02445=1012.500,-118.872,393.598,-156.582,87.213,-156.712
C02446=1012.499,-119.261,393.629,-158.451,87.123,-158.588
C02447=1012.500,-119.649,393.659,-160.219,87.030,-160.363
C02448=1012.501,-120.037,393.689,-161.875,86.935,-162.026
C02449=1012.501,-120.425,393.718,-163.427,86.837,-163.586
C02450=1012.501,-120.813,393.749,-164.900,86.735,-165.066
C02451=1012.502,-121.201,393.779,-166.280,86.632,-166.454
C02452=1012.503,-121.590,393.809,-167.591,86.525,-167.772
C02453=1012.502,-121.978,393.838,-168.833,86.417,-169.022
C02454=1012.502,-122.367,393.869,-169.987,86.307,-170.184
C02455=1012.503,-122.755,393.899,-171.094,86.195,-171.299
C02456=1012.503,-123.143,393.928,-172.126,86.081,-172.339
C02457=1012.504,-123.531,393.959,-173.108,85.965,-173.330
C02458=1012.505,-123.919,393.989,-174.042,85.848,-174.272
C02459=1012.506,-124.307,394.018,-174.923,85.729,-175.162
C02460=1012.506,-124.695,394.048,-175.764,85.608,-176.011
C02461=1012.506,-125.083,394.078,-176.557,85.487,-176.813
C02462=1012.507,-125.472,394.108,-177.306,85.365,-177.572
C02463=1012.508,-125.860,394.138,-178.023,85.240,-178.298
C02464=1012.507,-126.248,394.168,-178.709,85.114,-178.993
C02465=1012.508,-126.636,394.198,-179.358,84.987,-179.652
C02466=1012.509,-127.024,394.227,-179.981,84.859,179.716
C02467=1012.510,-127.412,394.258,179.429,84.730,179.117
C02468=1012.510,-127.800,394.288,178.869,84.601,178.547
C02469=1012.511,-128.189,394.317,178.331,84.469,177.999
C02470=1012.512,-128.576,394.347,177.814,84.337,177.472
C02471=1012.513,-128.964,394.377,177.322,84.204,176.970
C02472=1012.513,-129.353,394.407,176.854,84.071,176.492
C02473=1012.514,-129.740,394.436,176.398,83.935,176.025
C02474=1012.514,-130.128,394.467,175.970,83.799,175.586
C02475=1012.516,-130.516,394.496,175.556,83.663,175.161
C02476=1012.516,-130.904,394.526,175.156,83.525,174.751
C02477=1012.518,-131.291,394.556,174.777,83.386,174.359
C02478=1012.519,-131.680,394.586,174.408,83.247,173.979
C02479=1012.519,-132.068,394.616,174.057,83.107,173.617
C02480=1012.520,-132.455,394.646,173.721,82.967,173.269
C02481=1012.521,-132.843,394.675,173.392,82.825,172.929
C02482=1012.522,-133.231,394.705,173.081,82.684,172.606
C02483=1012.523,-133.619,394.734,172.780,82.541,172.293
C02484=1012.524,-134.007,394.765,172.489,82.397,171.989
C02485=1012.498,-134.032,394.333,-74.170,87.345,-74.136
C02486=1012.498,-133.645,394.303,-71.703,87.242,-71.665
C02487=1012.498,-133.257,394.273,-69.417,87.134,-69.374
C02488=1012.498,-132.869,394.243,-67.306,87.023,-67.259
C02489=1012.498,-132.481,394.213,-65.363,86.908,-65.312
C02490=1012.499,-132.093,394.183,-63.566,86.791,-63.511
C02491=1012.499,-131.706,394.153,-61.898,86.670,-61.839
C02492=1012.499,-131.318,394.122,-60.360,86.547,-60.297
C02493=1012.499,-130.930,394.093,-58.931,86.423,-58.865
C02494=1012.499,-130.541,394.062,-57.601,86.296,-57.531
C02495=1012.500,-130.154,394.033,-56.369,86.168,-56.296
C02496=1012.499,-129.766,394.002,-55.221,86.040,-55.145
C02497=1012.500,-129.378,393.972,-54.145,85.909,-54.067
C02498=1012.500,-128.990,393.942,-53.147,85.778,-53.065
C02499=1012.500,-128.602,393.912,-52.209,85.646,-52.125
C02500=1012.501,-128.214,393.881,-51.328,85.513,-51.241
C02501=1012.501,-127.826,393.851,-50.506,85.380,-50.417
C02502=1012.501,-127.438,393.821,-49.731,85.247,-49.640
C02503=1012.502,-127.050,393.791,-49.006,85.113,-48.913
C02504=1012.502,-126.662,393.761,-48.314,84.978,-48.219
C02505=1012.502,-126.274,393.730,-47.666,84.844,-47.568
C02506=1012.503,-125.886,393.700,-47.056,84.709,-46.957
C02507=1012.503,-125.498,393.670,-46.472,84.574,-46.371
C02508=1012.503,-125.110,393.640,-45.928,84.439,-45.826
C02509=1012.505,-124.722,393.610,-45.405,84.304,-45.301
C02510=1012.505,-124.334,393.580,-44.911,84.170,-44.806
C02511=1012.505,-123.946,393.550,-44.440,84.034,-44.335
C02512=1012.505,-123.558,393.519,-43.991,83.899,-43.885
C02513=1012.506,-123.169,393.489,-43.566,83.764,-43.459
C02514=1012.507,-122.781,393.459,-43.159,83.630,-43.050
C02515=1012.507,-122.394,393.429,-42.774,83.496,-42.665
C02516=1012.508,-122.005,393.399,-42.405,83.362,-42.295
C02517=1012.508,-121.617,393.369,-42.050,83.228,-41.939
C02518=1012.509,-121.229,393.338,-41.713,83.094,-41.602
C02519=1012.509,-120.841,393.308,-41.390,82.960,-41.279
C02520=1012.510,-120.452,393.277,-41.082,82.828,-40.971
C02521=1012.510,-120.064,393.247,-40.785,82.696,-40.674
C02522=1012.511,-119.676,393.218,-40.502,82.564,-40.391
C02523=1012.512,-119.288,393.187,-40.226,82.431,-40.116
C02524=1012.512,-118.900,393.157,-39.967,82.300,-39.858
C02525=1012.513,-118.511,393.127,-39.712,82.169,-39.602
C02526=1012.514,-118.123,393.096,-39.470,82.038,-39.361
C02527=1012.515,-117.734,393.066,-39.238,81.908,-39.130
C02528=1012.515,-117.346,393.035,-39.014,81.778,-38.907
C02529=1012.515,-116.958,393.005,-38.797,81.649,-38.690
C02530=1012.516,-116.570,392.975,-38.586,81.519,-38.480
C02531=1012.517,-116.181,392.945,-38.387,81.392,-38.282
C02532=1012.518,-115.793,392.915,-38.192,81.262,-38.089
C02533=1012.518,-115.404,392.885,-38.004,81.135,-37.901
C02534=1012.519,-115.016,392.854,-37.821,81.008,-37.720
C02535=1012.521,-114.627,392.824,-37.647,80.882,-37.547
C02536=1012.521,-114.239,392.793,-37.478,80.755,-37.380
C02537=1012.522,-113.850,392.763,-37.315,80.630,-37.219
C02538=1012.522,-113.461,392.733,-37.156,80.505,-37.060
C02539=1012.523,-113.073,392.703,-37.002,80.379,-36.909
C02540=1012.524,-112.684,392.672,-36.852,80.256,-36.761
C02541=1012.525,-112.296,392.642,-36.708,80.132,-36.619
C02542=1012.526,-111.907,392.612,-36.569,80.009,-36.482
C02543=1012.527,-111.518,392.582,-36.434,79.886,-36.349
C02544=1012.527,-111.130,392.552,-36.301,79.764,-36.217
C02545=1012.528,-110.741,392.522,-36.173,79.642,-36.092
C02546=1012.529,-110.352,392.490,-36.050,79.522,-35.971
C02547=1012.530,-109.964,392.460,-35.930,79.401,-35.854
C02548=1012.531,-109.575,392.430,-35.813,79.281,-35.739
C02549=1012.532,-109.180,392.399,-35.697,79.160,-35.625
C02550=1012.533,-108.764,392.367,-35.578,79.033,-35.509
C02551=1012.534,-108.544,392.350,-35.519,78.966,-35.452
C02552=1012.534,-108.319,392.331,-35.456,78.898,-35.390
C02553=1012.535,-108.090,392.314,-35.395,78.828,-35.332
C02554=1012.535,-107.858,392.296,-35.333,78.758,-35.271
C02555=1012.536,-107.626,392.278,-35.274,78.689,-35.214
C02556=1012.536,-107.395,392.260,-35.215,78.620,-35.156
C02557=1012.537,-107.169,392.242,-35.158,78.552,-35.101
C02558=1012.536,-106.949,392.225,-35.103,78.486,-35.048
C02559=1012.537,-106.735,392.208,-35.051,78.422,-34.997
C02560=1012.538,-106.327,392.177,-34.952,78.301,-34.902
C02561=1012.539,-105.937,392.146,-34.861,78.186,-34.813
C02562=1012.540,-105.548,392.116,-34.773,78.072,-34.728
C02563=1012.541,-105.160,392.086,-34.687,77.958,-34.646
C02564=1012.542,-104.772,392.055,-34.603,77.846,-34.565
C02565=1012.543,-104.383,392.025,-34.521,77.734,-34.485
C02566=1012.544,-103.995,391.994,-34.442,77.622,-34.410
C02567=1012.545,-103.609,391.965,-34.366,77.512,-34.338
C02568=1012.546,-103.222,391.935,-34.290,77.403,-34.265
C02569=1012.547,-102.837,391.905,-34.216,77.293,-34.195
C02570=1012.547,-102.451,391.875,-34.144,77.184,-34.126
C02571=1012.548,-102.067,391.844,-34.074,77.077,-34.060
C02572=1012.549,-101.683,391.814,-34.006,76.970,-33.995
C02573=1012.550,-101.300,391.785,-33.939,76.865,-33.931
C02574=1012.551,-100.919,391.755,-33.875,76.760,-33.871
C02575=1012.553,-100.538,391.725,-33.811,76.656,-33.811
C02576=1012.553,-100.159,391.696,-33.750,76.553,-33.753
C02577=1012.555,-99.780,391.666,-33.690,76.449,-33.697
C02578=1012.556,-99.403,391.637,-33.632,76.349,-33.643
C02579=1012.556,-99.027,391.607,-33.574,76.247,-33.589
C02580=1012.557,-98.650,391.578,-33.518,76.148,-33.537
C02581=1012.558,-98.274,391.549,-33.463,76.048,-33.485
C02582=1012.559,-97.899,391.519,-33.410,75.950,-33.437
C02583=1012.560,-97.523,391.490,-33.357,75.851,-33.387
C02584=1012.561,-97.147,391.461,-33.307,75.755,-33.341
C02585=1012.562,-96.771,391.432,-33.256,75.657,-33.294
C02586=1012.563,-96.394,391.402,-33.207,75.561,-33.249
C02587=1012.564,-96.018,391.373,-33.158,75.465,-33.203
C02588=1012.565,-95.639,391.343,-33.111,75.370,-33.161
C02589=1012.566,-95.260,391.313,-33.063,75.274,-33.117
C02590=1012.566,-94.880,391.284,-33.017,75.179,-33.075
C02591=1012.568,-94.498,391.254,-32.973,75.085,-33.035
C02592=1012.569,-94.115,391.224,-32.928,74.990,-32.995
C02593=1012.570,-93.732,391.195,-32.885,74.896,-32.956
C02594=1012.571,-93.346,391.165,-32.842,74.802,-32.917
C02595=1012.572,-92.961,391.134,-32.799,74.710,-32.878
C02596=1012.573,-92.574,391.104,-32.759,74.616,-32.843
C02597=1012.574,-92.186,391.074,-32.718,74.524,-32.806
C02598=1012.574,-91.798,391.044,-32.677,74.433,-32.769
C02599=1012.576,-91.409,391.013,-32.639,74.341,-32.735
C02600=1012.576,-91.021,390.983,-32.600,74.251,-32.701
C02601=1012.578,-90.667,390.956,-32.565,74.169,-32.669
C02602=1012.578,-90.398,390.935,-32.540,74.107,-32.647
C02603=1012.579,-90.187,390.918,-32.519,74.059,-32.629
C02604=1012.580,-89.954,390.900,-32.498,74.005,-32.611
C02605=1012.580,-89.703,390.880,-32.475,73.949,-32.590
C02606=1012.581,-89.444,390.860,-32.452,73.890,-32.570
C02607=1012.582,-89.188,390.840,-32.428,73.832,-32.548
C02608=1012.582,-88.945,390.822,-32.406,73.778,-32.529
C02609=1012.582,-88.727,390.805,-32.387,73.729,-32.514
C02610=1012.584,-88.342,390.774,-32.353,73.644,-32.483
C02611=1012.584,-87.965,390.745,-32.321,73.561,-32.456
C02612=1012.586,-87.603,390.717,-32.292,73.482,-32.431
C02613=1012.586,-87.234,390.688,-32.261,73.402,-32.404
C02614=1012.588,-86.857,390.659,-32.230,73.322,-32.376
C02615=1012.588,-86.470,390.629,-32.200,73.239,-32.351
C02616=1012.589,-86.063,390.597,-32.168,73.153,-32.324
C02617=1012.590,-85.840,390.580,-32.151,73.106,-32.309
C02618=1012.590,-85.605,390.561,-32.133,73.057,-32.294
C02619=1012.591,-85.366,390.543,-32.115,73.007,-32.279
C02620=1012.591,-85.127,390.524,-32.098,72.958,-32.264
C02621=1012.592,-84.898,390.507,-32.081,72.911,-32.249
C02622=1012.593,-84.479,390.474,-32.051,72.825,-32.224
C02623=1012.595,-84.087,390.443,-32.022,72.746,-32.199
C02624=1012.595,-83.696,390.413,-31.995,72.668,-32.176
C02625=1012.596,-83.301,390.382,-31.968,72.589,-32.154
C02626=1012.597,-82.903,390.351,-31.941,72.511,-32.131
C02627=1012.598,-82.508,390.321,-31.916,72.433,-32.111
C02628=1012.599,-82.109,390.289,-31.890,72.356,-32.089
C02629=1012.599,-81.711,390.258,-31.865,72.280,-32.069
C02630=1012.600,-81.313,390.227,-31.840,72.205,-32.047
C02631=1012.601,-80.917,390.196,-31.816,72.130,-32.028
C02632=1012.603,-80.519,390.165,-31.791,72.057,-32.007
C02633=1012.603,-80.120,390.134,-31.768,71.984,-31.987
C02634=1012.605,-79.720,390.103,-31.745,71.911,-31.968
C02635=1012.605,-79.320,390.072,-31.722,71.838,-31.950
C02636=1012.606,-78.920,390.041,-31.699,71.766,-31.931
C02637=1012.607,-78.520,390.009,-31.678,71.696,-31.914
C02638=1012.608,-78.118,389.979,-31.656,71.626,-31.896
C02639=1012.608,-77.717,389.948,-31.635,71.557,-31.879
C02640=1012.609,-77.315,389.916,-31.614,71.488,-31.863
C02641=1012.611,-76.913,389.885,-31.593,71.419,-31.845
C02642=1012.612,-76.511,389.854,-31.573,71.352,-31.829
C02643=1012.612,-76.108,389.823,-31.553,71.286,-31.813
C02644=1012.613,-75.705,389.791,-31.533,71.220,-31.797
C02645=1012.614,-75.302,389.760,-31.515,71.155,-31.783
C02646=1012.615,-74.900,389.729,-31.495,71.091,-31.767
C02647=1012.616,-74.497,389.697,-31.477,71.027,-31.753
C02648=1012.616,-74.093,389.666,-31.459,70.964,-31.739
C02649=1012.618,-73.690,389.634,-31.441,70.902,-31.725
C02650=1012.618,-73.286,389.602,-31.423,70.841,-31.709
C02651=1012.619,-72.883,389.572,-31.406,70.780,-31.695
C02652=1012.619,-72.479,389.540,-31.390,70.721,-31.683
C02653=1012.621,-72.075,389.509,-31.373,70.661,-31.671
C02654=1012.621,-71.671,389.477,-31.357,70.602,-31.657
C02655=1012.622,-71.267,389.446,-31.340,70.545,-31.643
C02656=1012.623,-70.863,389.415,-31.325,70.488,-31.632
C02657=1012.624,-70.459,389.383,-31.309,70.432,-31.619
C02658=1012.624,-70.054,389.352,-31.294,70.377,-31.608
C02659=1012.625,-69.650,389.320,-31.279,70.322,-31.596
C02660=1012.625,-69.246,389.289,-31.264,70.269,-31.584
C02661=1012.627,-68.842,389.258,-31.250,70.217,-31.573
C02662=1012.628,-68.437,389.226,-31.236,70.164,-31.562
C02663=1012.628,-68.033,389.195,-31.222,70.113,-31.550
C02664=1012.628,-67.629,389.163,-31.209,70.063,-31.541
C02665=1012.629,-67.225,389.133,-31.196,70.012,-31.530
C02666=1012.630,-66.821,389.100,-31.183,69.964,-31.520
C02667=1012.631,-66.417,389.069,-31.170,69.914,-31.510
C02668=1012.631,-66.014,389.038,-31.158,69.868,-31.500
C02669=1012.632,-65.610,389.006,-31.145,69.821,-31.491
C02670=1012.633,-65.208,388.975,-31.133,69.776,-31.481
C02671=1012.634,-64.805,388.944,-31.121,69.731,-31.471
C02672=1012.634,-64.403,388.912,-31.110,69.686,-31.463
C02673=1012.634,-64.001,388.881,-31.099,69.643,-31.453
C02674=1012.635,-63.598,388.850,-31.088,69.600,-31.445
C02675=1012.636,-63.198,388.820,-31.076,69.558,-31.435
C02676=1012.636,-62.797,388.788,-31.066,69.517,-31.427
C02677=1012.636,-62.396,388.757,-31.055,69.477,-31.418
C02678=1012.637,-61.997,388.726,-31.045,69.438,-31.409
C02679=1012.638,-61.598,388.695,-31.035,69.399,-31.402
C02680=1012.639,-61.199,388.663,-31.026,69.362,-31.395
C02681=1012.639,-60.800,388.633,-31.016,69.325,-31.387
C02682=1012.640,-60.402,388.603,-31.006,69.289,-31.378
C02683=1012.640,-60.005,388.571,-30.997,69.253,-31.370
C02684=1012.641,-59.608,388.540,-30.988,69.218,-31.364
C02685=1012.641,-59.212,388.510,-30.979,69.184,-31.356
C02686=1012.641,-58.816,388.479,-30.971,69.151,-31.349
C02687=1012.642,-58.421,388.448,-30.963,69.120,-31.343
C02688=1012.642,-58.026,388.418,-30.955,69.088,-31.336
C02689=1012.642,-57.632,388.387,-30.947,69.057,-31.329
C02690=1012.643,-57.238,388.356,-30.939,69.027,-31.322
C02691=1012.643,-56.845,388.326,-30.931,68.998,-31.316
C02692=1012.644,-56.451,388.295,-30.924,68.970,-31.309
C02693=1012.644,-56.058,388.265,-30.917,68.942,-31.303
C02694=1012.644,-55.666,388.235,-30.909,68.915,-31.297
C02695=1012.645,-55.274,388.204,-30.903,68.889,-31.291
C02696=1012.645,-54.881,388.174,-30.896,68.864,-31.286
C02697=1012.646,-54.488,388.143,-30.889,68.839,-31.278
C02698=1012.645,-54.096,388.113,-30.883,68.816,-31.273
C02699=1012.646,-53.703,388.082,-30.877,68.792,-31.267
C02700=1012.647,-53.311,388.052,-30.870,68.770,-31.261
C02701=1012.647,-52.919,388.022,-30.864,68.748,-31.255
C02702=1012.647,-52.526,387.991,-30.859,68.727,-31.251
C02703=1012.647,-52.133,387.961,-30.853,68.707,-31.245
C02704=1012.648,-51.741,387.930,-30.848,68.687,-31.239
C02705=1012.647,-51.348,387.900,-30.842,68.668,-31.235
C02706=1012.648,-50.956,387.869,-30.838,68.650,-31.230
C02707=1012.649,-50.563,387.839,-30.833,68.632,-31.225
C02708=1012.648,-50.171,387.809,-30.828,68.616,-31.220
C02709=1012.649,-49.778,387.778,-30.823,68.600,-31.215
C02710=1012.649,-49.386,387.748,-30.818,68.584,-31.210
C02711=1012.649,-48.992,387.717,-30.814,68.570,-31.206
C02712=1012.649,-48.600,387.687,-30.809,68.556,-31.200
C02713=1012.649,-48.207,387.656,-30.806,68.543,-31.197
C02714=1012.649,-47.814,387.626,-30.802,68.530,-31.191
C02715=1012.650,-47.422,387.595,-30.798,68.519,-31.188
C02716=1012.649,-47.029,387.565,-30.794,68.508,-31.182
C02717=1012.650,-46.636,387.535,-30.791,68.498,-31.179
C02718=1012.650,-46.244,387.504,-30.787,68.488,-31.174
C02719=1012.650,-45.851,387.474,-30.784,68.480,-31.170
C02720=1012.650,-45.457,387.444,-30.781,68.472,-31.166
C02721=1012.649,-45.065,387.413,-30.778,68.464,-31.162
C02722=1012.650,-44.672,387.382,-30.775,68.458,-31.158
C02723=1012.650,-44.279,387.352,-30.772,68.451,-31.153
C02724=1012.650,-43.886,387.322,-30.770,68.446,-31.150
C02725=1012.650,-43.493,387.292,-30.768,68.442,-31.147
C02726=1012.650,-43.099,387.261,-30.766,68.438,-31.144
C02727=1012.650,-42.707,387.230,-30.764,68.434,-31.140
C02728=1012.650,-42.314,387.199,-30.762,68.432,-31.137
C02729=1012.650,-41.921,387.169,-30.759,68.430,-31.131
C02730=1012.649,-41.528,387.139,-30.758,68.429,-31.129
C02731=1012.649,-41.135,387.109,-30.757,68.429,-31.126
C02732=1012.650,-40.742,387.078,-30.755,68.429,-31.123
C02733=1012.649,-40.348,387.047,-30.753,68.430,-31.119
C02734=1012.649,-39.955,387.017,-30.753,68.433,-31.117
C02735=1012.649,-39.562,386.987,-30.752,68.434,-31.114
C02736=1012.649,-39.168,386.956,-30.751,68.438,-31.111
C02737=1012.649,-38.775,386.926,-30.750,68.442,-31.108
C02738=1012.649,-38.381,386.895,-30.749,68.447,-31.104
C02739=1012.649,-37.988,386.864,-30.749,68.451,-31.102
C02740=1012.649,-37.594,386.835,-30.749,68.459,-31.099
C02741=1012.648,-37.201,386.804,-30.749,68.464,-31.097
C02742=1012.648,-36.808,386.774,-30.748,68.472,-31.094
C02743=1012.648,-36.414,386.743,-30.749,68.480,-31.092
C02744=1012.648,-36.021,386.713,-30.749,68.489,-31.089
C02745=1012.647,-35.628,386.682,-30.749,68.499,-31.087
C02746=1012.648,-35.234,386.652,-30.750,68.509,-31.085
C02747=1012.647,-34.840,386.622,-30.750,68.519,-31.083
C02748=1012.646,-34.447,386.591,-30.752,68.531,-31.082
C02749=1012.646,-34.054,386.560,-30.752,68.544,-31.078
C02750=1012.646,-33.660,386.530,-30.753,68.556,-31.077
C02751=1012.646,-33.267,386.499,-30.755,68.570,-31.075
C02752=1012.645,-32.873,386.469,-30.755,68.585,-31.072
C02753=1012.645,-32.480,386.439,-30.758,68.599,-31.072
C02754=1012.645,-32.087,386.408,-30.759,68.615,-31.070
C02755=1012.644,-31.693,386.377,-30.761,68.632,-31.068
C02756=1012.644,-31.299,386.348,-30.762,68.649,-31.066
C02757=1012.643,-30.906,386.317,-30.765,68.667,-31.065
C02758=1012.643,-30.512,386.286,-30.767,68.685,-31.064
C02759=1012.643,-30.119,386.256,-30.769,68.704,-31.062
C02760=1012.642,-29.725,386.226,-30.772,68.725,-31.062
C02761=1012.642,-29.332,386.196,-30.774,68.744,-31.061
C02762=1012.642,-28.939,386.165,-30.777,68.766,-31.059
C02763=1012.641,-28.545,386.134,-30.780,68.788,-31.059
C02764=1012.640,-28.152,386.105,-30.783,68.811,-31.057
C02765=1012.640,-27.759,386.074,-30.786,68.834,-31.056
C02766=1012.639,-27.365,386.043,-30.789,68.858,-31.056
C02767=1012.639,-26.972,386.013,-30.793,68.882,-31.055
C02768=1012.639,-26.579,385.982,-30.797,68.908,-31.056
C02769=1012.638,-26.185,385.952,-30.800,68.933,-31.055
C02770=1012.637,-25.792,385.922,-30.804,68.960,-31.054
C02771=1012.637,-25.399,385.891,-30.808,68.988,-31.054
C02772=1012.636,-25.005,385.860,-30.812,69.015,-31.054
C02773=1012.635,-24.611,385.830,-30.817,69.044,-31.056
C02774=1012.635,-24.219,385.800,-30.822,69.073,-31.055
C02775=1012.634,-23.825,385.769,-30.826,69.104,-31.054
C02776=1012.634,-23.432,385.739,-30.831,69.134,-31.055
C02777=1012.633,-23.039,385.709,-30.836,69.165,-31.056
C02778=1012.632,-22.645,385.679,-30.841,69.197,-31.057
C02779=1012.632,-22.252,385.648,-30.846,69.230,-31.056
C02780=1012.631,-21.859,385.617,-30.851,69.263,-31.057
C02781=1012.631,-21.466,385.587,-30.858,69.297,-31.059
C02782=1012.630,-21.073,385.556,-30.864,69.332,-31.061
C02783=1012.629,-20.679,385.526,-30.869,69.367,-31.061
C02784=1012.628,-20.283,385.496,-30.875,69.403,-31.061
C02785=1012.627,-19.932,385.469,-30.881,69.436,-31.064
C02786=1012.627,-19.727,385.452,-30.884,69.454,-31.064
C02787=1012.627,-19.497,385.435,-30.888,69.476,-31.065
C02788=1012.627,-19.240,385.415,-30.892,69.501,-31.066
C02789=1012.626,-18.965,385.394,-30.897,69.528,-31.068
C02790=1012.626,-18.687,385.372,-30.902,69.555,-31.068
C02791=1012.625,-18.414,385.351,-30.907,69.582,-31.070
C02792=1012.624,-18.161,385.332,-30.911,69.608,-31.071
C02793=1012.624,-17.935,385.315,-30.915,69.631,-31.073
C02794=1012.624,-17.538,385.284,-30.922,69.672,-31.074
C02795=1012.622,-17.149,385.253,-30.931,69.712,-31.078
C02796=1012.622,-16.751,385.223,-30.937,69.754,-31.079
C02797=1012.621,-16.354,385.192,-30.946,69.797,-31.083
C02798=1012.620,-15.958,385.162,-30.954,69.840,-31.086
C02799=1012.619,-15.564,385.131,-30.963,69.884,-31.090
C02800=1012.619,-15.176,385.101,-30.971,69.927,-31.092
C02801=1012.617,-14.796,385.072,-30.979,69.970,-31.095
C02802=1012.617,-14.422,385.043,-30.987,70.014,-31.099
C02803=1012.615,-14.046,385.014,-30.996,70.059,-31.101
C02804=1012.615,-13.665,384.985,-31.004,70.104,-31.105
C02805=1012.614,-13.272,384.954,-31.014,70.151,-31.108
C02806=1012.613,-12.867,384.923,-31.024,70.201,-31.113
C02807=1012.612,-12.455,384.891,-31.034,70.252,-31.117
C02808=1012.611,-12.042,384.859,-31.045,70.304,-31.123
C02809=1012.610,-11.626,384.827,-31.055,70.357,-31.127
C02810=1012.609,-11.209,384.795,-31.066,70.410,-31.133
C02811=1012.608,-10.790,384.763,-31.078,70.465,-31.139
C02812=1012.607,-10.371,384.730,-31.089,70.520,-31.144
C02813=1012.606,-9.951,384.698,-31.101,70.577,-31.150
C02814=1012.605,-9.529,384.666,-31.114,70.634,-31.157
C02815=1012.604,-9.106,384.633,-31.126,70.692,-31.164
C02816=1012.603,-8.896,384.617,-31.132,70.720,-31.167
C02817=1012.603,-8.685,384.601,-31.139,70.750,-31.169
C02818=1012.602,-8.473,384.584,-31.145,70.779,-31.174
C02819=1012.601,-8.262,384.568,-31.152,70.810,-31.178
C02820=1012.601,-8.050,384.551,-31.159,70.840,-31.180
C02821=1012.601,-7.838,384.535,-31.165,70.870,-31.183
C02822=1012.601,-7.625,384.519,-31.172,70.901,-31.187
C02823=1012.600,-7.411,384.502,-31.179,70.931,-31.192
C02824=1012.599,-7.197,384.485,-31.186,70.962,-31.196
C02825=1012.599,-6.982,384.469,-31.193,70.994,-31.200
C02826=1012.598,-6.766,384.452,-31.200,71.025,-31.204
C02827=1012.597,-6.551,384.436,-31.208,71.057,-31.208
C02828=1012.596,-6.334,384.419,-31.215,71.090,-31.212
C02829=1012.596,-6.117,384.402,-31.223,71.122,-31.217
C02830=1012.596,-5.900,384.385,-31.230,71.155,-31.221
C02831=1012.595,-5.683,384.369,-31.238,71.188,-31.227
C02832=1012.594,-5.467,384.352,-31.245,71.221,-31.229
C02833=1012.594,-5.252,384.336,-31.253,71.254,-31.235
C02834=1012.593,-4.838,384.303,-31.268,71.317,-31.244
C02835=1012.591,-4.448,384.273,-31.283,71.378,-31.254
C02836=1012.590,-4.068,384.244,-31.297,71.437,-31.262
C02837=1012.590,-3.683,384.214,-31.312,71.499,-31.270
C02838=1012.589,-3.280,384.184,-31.328,71.563,-31.281
C02839=1012.587,-2.869,384.152,-31.345,71.630,-31.292
C02840=1012.586,-2.459,384.120,-31.361,71.697,-31.303
C02841=1012.585,-2.050,384.088,-31.378,71.764,-31.314
C02842=1012.584,-1.644,384.058,-31.395,71.832,-31.324
C02843=1012.582,-1.240,384.026,-31.413,71.899,-31.337
C02844=1012.581,-0.838,383.995,-31.431,71.968,-31.349
C02845=1012.580,-0.437,383.964,-31.448,72.037,-31.360
C02846=1012.579,-0.039,383.934,-31.467,72.106,-31.374
C02847=1012.577,0.356,383.904,-31.485,72.174,-31.386
C02848=1012.576,0.751,383.873,-31.504,72.243,-31.400
C02849=1012.575,1.147,383.842,-31.523,72.314,-31.412
C02850=1012.574,1.544,383.812,-31.543,72.384,-31.426
C02851=1012.573,1.936,383.781,-31.563,72.455,-31.441
C02852=1012.572,2.307,383.753,-31.582,72.523,-31.456
C02853=1012.570,2.649,383.726,-31.600,72.585,-31.468
C02854=1012.570,2.973,383.702,-31.616,72.644,-31.480
C02855=1012.569,3.296,383.676,-31.634,72.704,-31.493
C02856=1012.567,3.641,383.650,-31.653,72.769,-31.507
C02857=1012.566,4.013,383.621,-31.674,72.838,-31.523
C02858=1012.565,4.403,383.591,-31.695,72.912,-31.539
C02859=1012.564,4.794,383.561,-31.718,72.986,-31.556
C02860=1012.562,5.182,383.532,-31.741,73.061,-31.574
C02861=1012.561,5.573,383.502,-31.764,73.136,-31.592
C02862=1012.560,5.965,383.472,-31.789,73.213,-31.612
C02863=1012.559,6.358,383.441,-31.812,73.290,-31.629
C02864=1012.557,6.749,383.410,-31.837,73.367,-31.649
C02865=1012.556,7.135,383.381,-31.861,73.443,-31.668
C02866=1012.554,7.516,383.352,-31.887,73.520,-31.689
C02867=1012.553,7.894,383.322,-31.912,73.596,-31.709
C02868=1012.552,8.271,383.294,-31.937,73.672,-31.729
C02869=1012.551,8.645,383.264,-31.963,73.748,-31.749
C02870=1012.550,9.018,383.235,-31.989,73.825,-31.772
C02871=1012.548,9.392,383.207,-32.016,73.903,-31.793
C02872=1012.547,9.766,383.178,-32.043,73.979,-31.816
C02873=1012.546,10.142,383.149,-32.070,74.059,-31.838
C02874=1012.545,10.520,383.121,-32.100,74.138,-31.863
C02875=1012.543,10.895,383.092,-32.129,74.218,-31.887
C02876=1012.541,11.260,383.064,-32.156,74.295,-31.910
C02877=1012.541,11.623,383.035,-32.186,74.373,-31.935
C02878=1012.539,11.995,383.008,-32.216,74.453,-31.960
C02879=1012.537,12.377,382.978,-32.247,74.535,-31.988
C02880=1012.537,12.762,382.948,-32.280,74.619,-32.016
C02881=1012.535,13.145,382.918,-32.313,74.703,-32.044
C02882=1012.534,13.528,382.890,-32.347,74.787,-32.075
C02883=1012.533,13.910,382.860,-32.381,74.873,-32.104
C02884=1012.531,14.291,382.830,-32.414,74.957,-32.132
C02885=1012.530,14.671,382.801,-32.451,75.042,-32.166
C02886=1012.529,15.051,382.772,-32.486,75.128,-32.197
C02887=1012.528,15.431,382.743,-32.523,75.214,-32.228
C02888=1012.526,15.812,382.714,-32.560,75.300,-32.262
C02889=1012.525,16.193,382.684,-32.598,75.389,-32.295
C02890=1012.523,16.576,382.655,-32.637,75.476,-32.330
C02891=1012.522,16.960,382.625,-32.678,75.566,-32.367
C02892=1012.520,17.346,382.596,-32.718,75.655,-32.404
C02893=1012.519,17.734,382.565,-32.761,75.746,-32.443
C02894=1012.517,18.124,382.536,-32.803,75.838,-32.480
C02895=1012.516,18.516,382.506,-32.848,75.930,-32.523
C02896=1012.515,18.915,382.475,-32.893,76.026,-32.562
C02897=1012.513,19.318,382.444,-32.942,76.121,-32.608
C02898=1012.512,19.521,382.428,-32.966,76.171,-32.631
C02899=1012.512,19.742,382.411,-32.993,76.224,-32.656
C02900=1012.510,19.985,382.392,-33.022,76.282,-32.681
C02901=1012.510,20.245,382.373,-33.054,76.346,-32.712
C02902=1012.509,20.514,382.352,-33.089,76.411,-32.744
C02903=1012.508,20.783,382.331,-33.123,76.476,-32.776
C02904=1012.507,21.044,382.312,-33.156,76.539,-32.807
C02905=1012.506,21.291,382.293,-33.189,76.601,-32.837
C02906=1012.505,21.519,382.275,-33.219,76.656,-32.866
C02907=1012.504,21.908,382.244,-33.273,76.752,-32.916
C02908=1012.503,22.236,382.220,-33.318,76.834,-32.959
C02909=1012.501,22.567,382.195,-33.364,76.916,-33.002
C02910=1012.500,22.844,382.173,-33.403,76.985,-33.039
C02911=1012.499,23.208,382.146,-33.457,77.076,-33.090
C02912=1012.497,23.624,382.113,-33.518,77.181,-33.148
C02913=1012.496,23.964,382.087,-33.571,77.268,-33.198
C02914=1012.495,24.344,382.058,-33.630,77.364,-33.254
C02915=1012.493,24.739,382.028,-33.692,77.465,-33.313
C02916=1012.491,25.135,381.997,-33.756,77.566,-33.375
C02917=1012.491,25.531,381.967,-33.822,77.668,-33.439
C02918=1012.489,25.930,381.936,-33.892,77.771,-33.506
C02919=1012.487,26.327,381.906,-33.961,77.874,-33.573
C02920=1012.486,26.724,381.875,-34.031,77.977,-33.641
C02921=1012.485,27.119,381.845,-34.104,78.082,-33.711
C02922=1012.484,27.512,381.815,-34.177,78.185,-33.782
C02923=1012.482,27.905,381.785,-34.252,78.289,-33.855
C02924=1012.480,28.298,381.754,-34.330,78.392,-33.931
C02925=1012.479,28.691,381.724,-34.409,78.498,-34.008
C02926=1012.477,29.087,381.694,-34.491,78.603,-34.088
C02927=1012.475,29.482,381.664,-34.575,78.709,-34.171
C02928=1012.474,29.877,381.633,-34.660,78.816,-34.254
C02929=1012.473,30.273,381.602,-34.750,78.923,-34.343
C02930=1012.471,30.668,381.572,-34.841,79.031,-34.432
C02931=1012.470,31.064,381.542,-34.934,79.139,-34.523
C02932=1012.468,31.459,381.512,-35.028,79.246,-34.617
C02933=1012.467,31.854,381.481,-35.126,79.355,-34.713
C02934=1012.466,32.250,381.450,-35.226,79.464,-34.812
C02935=1012.464,32.644,381.421,-35.331,79.574,-34.916
C02936=1012.463,33.040,381.391,-35.437,79.683,-35.022
C02937=1012.462,33.436,381.360,-35.546,79.794,-35.129
C02938=1012.460,33.831,381.330,-35.659,79.905,-35.242
C02939=1012.459,34.226,381.299,-35.774,80.016,-35.358
C02940=1012.457,34.622,381.269,-35.892,80.127,-35.474
C02941=1012.456,35.017,381.238,-36.015,80.239,-35.597
C02942=1012.454,35.412,381.208,-36.140,80.352,-35.722
C02943=1012.453,35.808,381.178,-36.269,80.464,-35.851
C02944=1012.451,36.204,381.148,-36.403,80.577,-35.985
C02945=1012.450,36.600,381.117,-36.540,80.690,-36.122
C02946=1012.448,36.994,381.087,-36.681,80.804,-36.263
C02947=1012.447,37.390,381.056,-36.828,80.917,-36.411
C02948=1012.446,37.785,381.026,-36.978,81.032,-36.562
C02949=1012.444,38.181,380.996,-37.133,81.146,-36.716
C02950=1012.443,38.576,380.966,-37.294,81.261,-36.879
C02951=1012.441,38.972,380.935,-37.459,81.377,-37.044
C02952=1012.440,39.368,380.905,-37.628,81.493,-37.214
C02953=1012.439,39.763,380.874,-37.806,81.609,-37.393
C02954=1012.437,40.159,380.844,-37.988,81.725,-37.577
C02955=1012.436,40.555,380.814,-38.176,81.842,-37.765
C02956=1012.434,40.950,380.784,-38.372,81.959,-37.963
C02957=1012.433,41.345,380.753,-38.574,82.076,-38.167
C02958=1012.432,41.741,380.722,-38.782,82.194,-38.376
C02959=1012.430,42.137,380.692,-39.000,82.311,-38.597
C02960=1012.429,42.532,380.661,-39.225,82.429,-38.824
C02961=1012.428,42.928,380.631,-39.456,82.548,-39.056
C02962=1012.426,43.324,380.601,-39.700,82.666,-39.303
C02963=1012.425,43.719,380.570,-39.951,82.785,-39.556
C02964=1012.424,44.115,380.540,-40.211,82.904,-39.818
C02965=1012.422,44.511,380.510,-40.479,83.024,-40.088
C02966=1012.421,44.907,380.479,-40.761,83.144,-40.372
C02967=1012.420,45.302,380.449,-41.057,83.264,-40.672
C02968=1012.418,45.698,380.419,-41.360,83.383,-40.978
C02969=1012.417,46.094,380.388,-41.679,83.504,-41.299
C02970=1012.416,46.490,380.358,-42.010,83.623,-41.635
C02971=1012.414,46.885,380.327,-42.358,83.745,-41.985
C02972=1012.413,47.281,380.297,-42.716,83.864,-42.347
C02973=1012.412,47.677,380.267,-43.098,83.986,-42.732
C02974=1012.410,48.073,380.236,-43.491,84.106,-43.129
C02975=1012.409,48.468,380.206,-43.905,84.227,-43.548
C02976=1012.408,48.864,380.176,-44.338,84.348,-43.984
C02977=1012.407,49.260,380.145,-44.790,84.468,-44.441
C02978=1012.405,49.657,380.115,-45.268,84.590,-44.923
C02979=1012.404,50.053,380.085,-45.769,84.710,-45.428
C02980=1012.402,50.448,380.054,-46.293,84.831,-45.957
C02981=1012.401,50.844,380.024,-46.849,84.952,-46.518
C02982=1012.400,51.240,379.993,-47.427,85.072,-47.100
C02983=1012.399,51.636,379.963,-48.040,85.191,-47.719
C02984=1012.398,52.032,379.933,-48.693,85.312,-48.377
C02985=1012.396,52.428,379.902,-49.373,85.431,-49.062
C02986=1012.396,52.824,379.872,-50.097,85.550,-49.792
C02987=1012.394,53.220,379.841,-50.862,85.668,-50.562
C02988=1012.393,53.616,379.811,-51.679,85.787,-51.385
C02989=1012.392,54.012,379.780,-52.536,85.904,-52.247
C02990=1012.391,54.408,379.750,-53.452,86.020,-53.170
C02991=1012.389,54.804,379.720,-54.425,86.136,-54.149
C02992=1012.389,55.201,379.689,-55.468,86.251,-55.198
C02993=1012.387,55.596,379.659,-56.568,86.365,-56.304
C02994=1012.387,55.992,379.629,-57.749,86.477,-57.492
C02995=1012.386,56.388,379.598,-59.021,86.589,-58.772
C02996=1012.385,56.784,379.568,-60.369,86.698,-60.126
C02997=1012.384,57.180,379.537,-61.820,86.806,-61.585
C02998=1012.382,57.576,379.507,-63.372,86.911,-63.145
C02999=1012.381,57.972,379.477,-65.039,87.015,-64.818
C03000=1012.380,58.368,379.446,-66.824,87.116,-66.611
C03001=1012.379,58.765,379.416,-68.751,87.214,-68.546
C03002=1012.378,59.161,379.385,-70.825,87.309,-70.627
C03003=1012.377,59.557,379.355,-73.047,87.401,-72.858
C03004=1012.376,59.953,379.324,-75.428,87.488,-75.247
C03005=1012.375,60.349,379.294,-77.993,87.570,-77.820
C03006=1012.374,60.745,379.263,-80.744,87.648,-80.579
C03007=1012.373,61.141,379.233,-83.675,87.720,-83.519
C03008=1012.372,61.538,379.202,-86.788,87.785,-86.641
C03009=1012.371,61.933,379.172,-90.116,87.844,-89.978
C03010=1012.370,62.332,379.142,-93.638,87.896,-93.509
C03011=1012.370,62.615,379.120,-96.229,87.927,-96.107
C03012=1012.369,62.835,379.103,-98.318,87.949,-98.201
C03013=1012.368,63.077,379.084,-100.656,87.969,-100.545
C03014=1012.368,63.325,379.065,-103.080,87.986,-102.975
C03015=1012.367,63.561,379.047,-105.433,87.999,-105.333
C03016=1012.367,63.772,379.031,-107.595,88.008,-107.501
C03017=1012.365,64.177,378.995,-108.727,88.012,-108.635
C03018=1012.365,64.396,378.974,-108.879,88.012,-108.787
C03019=1012.364,64.623,378.953,-109.011,88.013,-108.919
C03020=1012.364,64.849,378.932,-109.164,88.013,-109.072
C03021=1012.364,65.072,378.911,-109.296,88.014,-109.204
C03022=1012.363,65.291,378.891,-109.448,88.014,-109.357
C03023=1012.363,65.505,378.870,-109.581,88.015,-109.489
C03024=1012.362,65.713,378.851,-109.689,88.015,-109.598
C03025=1012.361,66.107,378.814,-109.954,88.016,-109.863
C03026=1012.360,66.433,378.784,-110.151,88.016,-110.060
C03027=1012.359,66.798,378.750,-110.392,88.017,-110.301
C03028=1012.358,67.195,378.712,-110.658,88.018,-110.566
C03029=1012.357,67.592,378.675,-110.919,88.018,-110.829
C03030=1012.356,67.994,378.638,-111.185,88.019,-111.095
C03031=1012.355,68.405,378.599,-111.447,88.019,-111.357
C03032=1012.353,68.823,378.560,-111.713,88.020,-111.623
C03033=1012.353,69.239,378.521,-111.999,88.020,-111.910
C03034=1012.352,69.647,378.483,-112.286,88.021,-112.196
C03035=1012.351,70.051,378.445,-112.528,88.021,-112.439
C03036=1012.350,70.456,378.407,-112.815,88.021,-112.726
C03037=1012.349,70.860,378.369,-113.081,88.022,-112.992
C03038=1012.348,71.266,378.330,-113.344,88.022,-113.255
C03039=1012.346,71.670,378.293,-113.630,88.022,-113.542
C03040=1012.346,72.075,378.254,-113.897,88.022,-113.809
C03041=1012.344,72.481,378.216,-114.184,88.022,-114.096
C03042=1012.344,72.889,378.178,-114.446,88.022,-114.359
C03043=1012.343,73.298,378.139,-114.733,88.022,-114.646
C03044=1012.341,73.709,378.101,-115.000,88.022,-114.913
C03045=1012.341,74.125,378.061,-115.287,88.022,-115.200
C03046=1012.339,74.344,378.041,-115.440,88.022,-115.353
C03047=1012.339,74.573,378.019,-115.618,88.022,-115.531
C03048=1012.338,74.799,377.998,-115.771,88.022,-115.685
C03049=1012.338,75.015,377.977,-115.905,88.022,-115.818
C03050=1012.337,75.223,377.958,-116.058,88.021,-115.972
C03051=1012.336,75.637,377.918,-116.344,88.021,-116.258
C03052=1012.335,76.046,377.880,-116.631,88.021,-116.545
C03053=1012.334,76.449,377.842,-116.917,88.020,-116.831
C03054=1012.333,76.842,377.805,-117.203,88.020,-117.118
C03055=1012.332,77.228,377.768,-117.444,88.019,-117.360
C03056=1012.331,77.611,377.731,-117.730,88.019,-117.646
C03057=1012.330,77.992,377.695,-117.971,88.018,-117.887
C03058=1012.329,78.375,377.659,-118.257,88.018,-118.173
C03059=1012.327,78.765,377.622,-118.542,88.017,-118.458
C03060=1012.326,79.160,377.585,-118.827,88.016,-118.744
C03061=1012.325,79.562,377.547,-119.112,88.015,-119.029
C03062=1012.324,79.970,377.508,-119.396,88.015,-119.313
C03063=1012.322,80.383,377.469,-119.681,88.014,-119.598
C03064=1012.322,80.766,377.432,-119.965,88.013,-119.882
C03065=1012.321,81.129,377.397,-120.223,88.011,-120.141
C03066=1012.320,81.523,377.361,-120.506,88.010,-120.425
C03067=1012.319,81.938,377.320,-120.789,88.009,-120.708
C03068=1012.317,82.352,377.281,-121.116,88.008,-121.035
C03069=1012.317,82.764,377.242,-121.398,88.007,-121.318
C03070=1012.315,83.177,377.202,-121.698,88.005,-121.619
C03071=1012.314,83.587,377.163,-121.980,88.004,-121.900
C03072=1012.313,83.997,377.125,-122.305,88.002,-122.226
C03073=1012.312,84.405,377.085,-122.585,88.001,-122.507
C03074=1012.310,84.812,377.046,-122.865,88.000,-122.787
C03075=1012.309,85.219,377.008,-123.163,87.998,-123.086
C03076=1012.308,85.622,376.969,-123.468,87.996,-123.390
C03077=1012.307,86.025,376.931,-123.765,87.994,-123.688
C03078=1012.306,86.428,376.892,-124.043,87.993,-123.967
C03079=1012.304,86.828,376.854,-124.338,87.991,-124.263
C03080=1012.303,87.228,376.816,-124.642,87.989,-124.566
C03081=1012.302,87.621,376.778,-124.936,87.987,-124.861
C03082=1012.301,88.006,376.740,-125.212,87.985,-125.137
C03083=1012.300,88.383,376.705,-125.487,87.983,-125.413
C03084=1012.299,88.759,376.669,-125.763,87.981,-125.688
C03085=1012.297,89.136,376.632,-126.037,87.979,-125.963
C03086=1012.296,89.521,376.596,-126.328,87.977,-126.255
C03087=1012.296,89.917,376.558,-126.601,87.975,-126.529
C03088=1012.295,90.151,376.535,-126.746,87.973,-126.674
C03089=1012.294,90.427,376.508,-126.933,87.972,-126.862
C03090=1012.292,90.706,376.481,-127.120,87.970,-127.049
C03091=1012.292,90.952,376.457,-127.307,87.968,-127.236
C03092=1012.291,91.355,376.419,-127.621,87.966,-127.550
C03093=1012.290,91.750,376.381,-127.907,87.963,-127.838
C03094=1012.289,92.144,376.343,-128.219,87.960,-128.150
C03095=1012.288,92.539,376.305,-128.530,87.958,-128.461
C03096=1012.286,92.933,376.267,-128.815,87.955,-128.746
C03097=1012.285,93.328,376.229,-129.098,87.952,-129.031
C03098=1012.283,93.723,376.191,-129.365,87.949,-129.298
C03099=1012.283,94.118,376.152,-129.631,87.947,-129.564
C03100=1012.282,94.512,376.114,-129.896,87.944,-129.830
C03101=1012.280,94.907,376.077,-130.176,87.941,-130.111
C03102=1012.279,95.301,376.038,-130.481,87.938,-130.416
C03103=1012.278,95.696,376.000,-130.785,87.934,-130.721
C03104=1012.276,96.091,375.962,-131.063,87.931,-130.999
C03105=1012.275,96.485,375.924,-131.406,87.927,-131.343
C03106=1012.274,96.879,375.886,-131.682,87.924,-131.619
C03107=1012.273,97.273,375.847,-131.941,87.921,-131.879
C03108=1012.272,97.668,375.809,-132.215,87.917,-132.153
C03109=1012.270,98.063,375.771,-132.488,87.914,-132.427
C03110=1012.269,98.457,375.733,-132.785,87.910,-132.725
C03111=1012.268,98.852,375.695,-133.081,87.907,-133.021
C03112=1012.267,99.246,375.656,-133.365,87.902,-133.307
C03113=1012.265,99.640,375.619,-133.685,87.899,-133.626
C03114=1012.264,100.035,375.579,-133.992,87.894,-133.934
C03115=1012.263,100.430,375.541,-134.259,87.891,-134.202
C03116=1012.262,100.824,375.503,-134.510,87.887,-134.454
C03117=1012.261,101.218,375.464,-134.774,87.883,-134.719
C03118=1012.259,101.613,375.426,-135.063,87.879,-135.008
C03119=1012.258,102.007,375.388,-135.339,87.875,-135.286
C03120=1012.257,102.402,375.350,-135.626,87.870,-135.573
C03121=1012.255,102.796,375.311,-135.950,87.866,-135.897
C03122=1012.254,103.190,375.272,-136.261,87.861,-136.209
C03123=1012.253,103.585,375.234,-136.505,87.857,-136.454
C03124=1012.252,103.979,375.196,-136.762,87.852,-136.712
C03125=1012.250,104.373,375.157,-137.042,87.848,-136.992
C03126=1012.249,104.768,375.119,-137.297,87.844,-137.248
C03127=1012.248,105.162,375.080,-137.588,87.839,-137.540
C03128=1012.247,105.556,375.042,-137.878,87.834,-137.831
C03129=1012.246,105.950,375.003,-138.191,87.828,-138.144
C03130=1012.244,106.345,374.965,-138.478,87.823,-138.432
C03131=1012.243,106.739,374.926,-138.763,87.818,-138.719
C03132=1012.242,107.133,374.888,-138.998,87.814,-138.954
C03133=1012.240,107.528,374.849,-139.257,87.809,-139.214
C03134=1012.239,107.922,374.810,-139.526,87.804,-139.484
C03135=1012.237,108.317,374.772,-139.807,87.798,-139.765
C03136=1012.236,108.711,374.733,-140.086,87.793,-140.045
C03137=1012.235,109.105,374.695,-140.363,87.787,-140.324
C03138=1012.234,109.499,374.656,-140.663,87.782,-140.624
C03139=1012.233,109.893,374.617,-140.950,87.775,-140.912
C03140=1012.231,110.287,374.578,-141.187,87.770,-141.151
C03141=1012.230,110.681,374.540,-141.448,87.765,-141.412
C03142=1012.228,111.076,374.501,-141.707,87.760,-141.671
C03143=1012.227,111.470,374.462,-141.976,87.754,-141.941
C03144=1012.226,111.864,374.423,-142.243,87.748,-142.210
C03145=1012.225,112.259,374.384,-142.521,87.742,-142.489
C03146=1012.223,112.654,374.346,-142.809,87.735,-142.777
C03147=1012.223,113.048,374.307,-143.083,87.729,-143.053
C03148=1012.221,113.442,374.268,-143.334,87.723,-143.305
C03149=1012.220,113.836,374.230,-143.571,87.717,-143.543
C03150=1012.219,114.230,374.190,-143.820,87.712,-143.792
C03151=1012.218,114.624,374.151,-144.077,87.705,-144.051
C03152=1012.216,115.018,374.112,-144.334,87.699,-144.308
C03153=1012.215,115.412,374.074,-144.622,87.692,-144.597
C03154=1012.213,115.807,374.035,-144.885,87.685,-144.862
C03155=1012.212,116.201,373.996,-145.170,87.678,-145.148
C03156=1012.211,116.595,373.957,-145.420,87.671,-145.399
C03157=1012.209,116.989,373.918,-145.636,87.666,-145.616
C03158=1012.209,117.384,373.879,-145.883,87.659,-145.864
C03159=1012.207,117.779,373.840,-146.129,87.652,-146.111
C03160=1012.205,118.173,373.801,-146.396,87.646,-146.379
C03161=1012.205,118.566,373.762,-146.649,87.638,-146.633
C03162=1012.203,118.961,373.723,-146.922,87.631,-146.907
C03163=1012.201,119.355,373.684,-147.172,87.623,-147.158
C03164=1012.200,119.749,373.645,-147.441,87.616,-147.429
C03165=1012.199,120.143,373.606,-147.669,87.609,-147.657
C03166=1012.198,120.538,373.567,-147.883,87.603,-147.872
C03167=1012.197,120.932,373.527,-148.117,87.596,-148.108
C03168=1012.195,121.326,373.488,-148.381,87.588,-148.372
C03169=1012.194,121.720,373.449,-148.621,87.580,-148.614
C03170=1012.192,122.115,373.410,-148.881,87.572,-148.875
C03171=1012.191,122.509,373.372,-149.139,87.564,-149.135
C03172=1012.190,122.903,373.332,-149.396,87.556,-149.392
C03173=1012.189,123.298,373.292,-149.600,87.549,-149.598
C03174=1012.187,123.692,373.253,-149.824,87.542,-149.823
C03175=1012.186,124.085,373.214,-150.055,87.534,-150.055
C03176=1012.185,124.480,373.175,-150.297,87.526,-150.298
C03177=1012.184,124.875,373.136,-150.525,87.518,-150.528
C03178=1012.182,125.269,373.097,-150.772,87.510,-150.776
C03179=1012.180,125.663,373.057,-151.026,87.501,-151.031
C03180=1012.180,126.057,373.018,-151.269,87.493,-151.276
C03181=1012.178,126.452,372.979,-151.491,87.484,-151.499
C03182=1012.177,126.846,372.939,-151.703,87.477,-151.712
C03183=1012.175,127.240,372.900,-151.914,87.469,-151.924
C03184=1012.174,127.635,372.860,-152.152,87.461,-152.163
C03185=1012.173,128.029,372.821,-152.368,87.452,-152.380
C03186=1012.171,128.423,372.782,-152.602,87.444,-152.616
C03187=1012.170,128.818,372.741,-152.842,87.434,-152.858
C03188=1012.169,129.212,372.702,-153.080,87.425,-153.097
C03189=1012.168,129.606,372.664,-153.310,87.416,-153.328
C03190=1012.167,130.000,372.624,-153.511,87.408,-153.530
C03191=1012.165,130.395,372.585,-153.717,87.400,-153.738
C03192=1012.164,130.788,372.545,-153.923,87.391,-153.945
C03193=1012.163,131.183,372.505,-154.146,87.382,-154.170
C03194=1012.161,131.578,372.466,-154.368,87.373,-154.393
C03195=1012.161,131.972,372.426,-154.595,87.364,-154.621
C03196=1012.159,132.367,372.387,-154.820,87.354,-154.848
C03197=1012.157,132.760,372.347,-155.043,87.344,-155.073
C03198=1012.156,133.155,372.308,-155.234,87.336,-155.265
C03199=1012.154,133.549,372.267,-155.429,87.327,-155.462
C03200=1012.153,133.944,372.228,-155.642,87.318,-155.675
C03201=1012.152,134.338,372.188,-155.840,87.308,-155.876
C03202=1012.151,134.733,372.149,-156.050,87.299,-156.087
C03203=1012.150,134.963,372.125,-156.185,87.293,-156.223
C03204=1012.149,135.223,372.100,-156.319,87.286,-156.358
C03205=1012.148,135.633,372.058,-156.550,87.276,-156.590
C03206=1012.147,136.002,372.021,-156.760,87.266,-156.802
C03207=1012.146,136.343,371.987,-156.921,87.258,-156.965
C03208=1012.144,136.665,371.955,-157.094,87.250,-157.138
C03209=1012.144,136.985,371.922,-157.253,87.242,-157.299
C03210=1012.142,137.328,371.887,-157.429,87.234,-157.477
C03211=1012.141,137.677,371.852,-157.604,87.225,-157.653
C03212=1012.141,137.977,371.822,-157.760,87.217,-157.811
C03213=1012.139,138.373,371.783,-157.956,87.207,-158.008
C03214=1012.138,138.593,371.760,-158.059,87.202,-158.112
C03215=1012.138,138.828,371.736,-158.184,87.195,-158.238
C03216=1012.137,139.077,371.711,-158.304,87.189,-158.358
C03217=1012.136,139.334,371.685,-158.428,87.183,-158.483
C03218=1012.135,139.597,371.658,-158.557,87.176,-158.614
C03219=1012.134,139.858,371.632,-158.680,87.169,-158.738
C03220=1012.133,140.112,371.607,-158.802,87.162,-158.861
C03221=1012.133,140.354,371.582,-158.919,87.156,-158.979
C03222=1012.132,140.581,371.559,-159.040,87.150,-159.101
C03223=1012.131,140.792,371.538,-159.134,87.145,-159.195
C03224=1012.130,141.010,371.516,-159.232,87.139,-159.294
C03225=1012.129,141.415,371.474,-159.444,87.128,-159.508
C03226=1012.128,141.680,371.448,-159.562,87.121,-159.628
C03227=1012.127,141.880,371.428,-159.654,87.116,-159.721
C03228=1012.127,142.281,371.387,-159.846,87.105,-159.915
C03229=1012.125,142.683,371.346,-160.032,87.094,-160.102
C03230=1012.124,143.084,371.305,-160.216,87.084,-160.288
C03231=1012.122,143.487,371.264,-160.399,87.073,-160.473
C03232=1012.122,143.890,371.224,-160.597,87.062,-160.672
C03233=1012.120,144.294,371.183,-160.781,87.050,-160.859
C03234=1012.119,144.699,371.142,-160.960,87.040,-161.039
C03235=1012.117,145.103,371.101,-161.141,87.028,-161.223
C03236=1012.116,145.509,371.059,-161.317,87.017,-161.401
C03237=1012.115,145.914,371.018,-161.512,87.005,-161.597
C03238=1012.114,146.321,370.977,-161.685,86.994,-161.772
C03239=1012.112,146.727,370.936,-161.861,86.983,-161.950
C03240=1012.111,147.134,370.894,-162.048,86.971,-162.138
C03241=1012.122,147.089,370.456,-39.562,82.848,-39.026
C03242=1012.123,146.681,370.497,-39.532,82.834,-38.995
C03243=1012.124,146.275,370.539,-39.498,82.819,-38.960
C03244=1012.125,145.869,370.580,-39.468,82.804,-38.930
C03245=1012.127,145.463,370.622,-39.435,82.789,-38.896
C03246=1012.128,145.058,370.662,-39.405,82.775,-38.865
C03247=1012.129,144.653,370.703,-39.372,82.760,-38.831
C03248=1012.132,144.249,370.744,-39.342,82.746,-38.801
C03249=1012.132,143.845,370.785,-39.310,82.731,-38.768
C03250=1012.134,143.442,370.826,-39.279,82.717,-38.736
C03251=1012.135,143.039,370.868,-39.250,82.703,-38.706
C03252=1012.137,142.637,370.908,-39.221,82.689,-38.677
C03253=1012.138,142.235,370.949,-39.192,82.674,-38.648
C03254=1012.139,141.835,370.989,-39.160,82.659,-38.615
C03255=1012.140,141.635,371.009,-39.147,82.652,-38.602
C03256=1012.141,141.370,371.036,-39.129,82.643,-38.584
C03257=1012.142,140.964,371.077,-39.097,82.628,-38.551
C03258=1012.143,140.747,371.099,-39.081,82.621,-38.534
C03259=1012.144,140.536,371.121,-39.069,82.614,-38.522
C03260=1012.145,140.310,371.144,-39.049,82.606,-38.502
C03261=1012.146,140.067,371.168,-39.035,82.597,-38.487
C03262=1012.146,139.813,371.194,-39.017,82.588,-38.469
C03263=1012.147,139.552,371.220,-38.999,82.579,-38.451
C03264=1012.149,139.290,371.247,-38.981,82.570,-38.432
C03265=1012.149,139.032,371.272,-38.963,82.561,-38.414
C03266=1012.150,138.783,371.298,-38.945,82.552,-38.396
C03267=1012.151,138.547,371.322,-38.931,82.544,-38.382
C03268=1012.152,138.329,371.344,-38.915,82.536,-38.366
C03269=1012.153,137.933,371.384,-38.886,82.523,-38.336
C03270=1012.154,137.632,371.414,-38.866,82.512,-38.316
C03271=1012.155,137.283,371.449,-38.841,82.499,-38.290
C03272=1012.157,136.940,371.484,-38.818,82.488,-38.267
C03273=1012.157,136.619,371.516,-38.799,82.476,-38.249
C03274=1012.158,136.298,371.548,-38.777,82.465,-38.225
C03275=1012.159,135.958,371.583,-38.754,82.454,-38.202
C03276=1012.161,135.588,371.620,-38.730,82.440,-38.178
C03277=1012.163,135.179,371.661,-38.700,82.425,-38.147
C03278=1012.163,134.919,371.687,-38.683,82.416,-38.130
C03279=1012.164,134.688,371.710,-38.666,82.407,-38.112
C03280=1012.166,134.293,371.750,-38.641,82.394,-38.087
C03281=1012.167,133.899,371.790,-38.618,82.380,-38.064
C03282=1012.169,133.505,371.829,-38.593,82.367,-38.039
C03283=1012.170,133.111,371.869,-38.569,82.355,-38.014
C03284=1012.171,132.716,371.908,-38.545,82.342,-37.990
C03285=1012.172,132.322,371.948,-38.519,82.327,-37.963
C03286=1012.174,131.927,371.987,-38.492,82.313,-37.937
C03287=1012.175,131.534,372.027,-38.470,82.299,-37.914
C03288=1012.176,131.139,372.067,-38.443,82.286,-37.886
C03289=1012.179,130.744,372.106,-38.419,82.273,-37.862
C03290=1012.180,130.350,372.146,-38.396,82.259,-37.840
C03291=1012.181,129.955,372.186,-38.376,82.247,-37.819
C03292=1012.183,129.562,372.225,-38.354,82.235,-37.797
C03293=1012.184,129.167,372.264,-38.329,82.221,-37.771
C03294=1012.186,128.773,372.304,-38.307,82.207,-37.750
C03295=1012.187,128.378,372.344,-38.280,82.194,-37.722
C03296=1012.188,127.984,372.383,-38.258,82.180,-37.700
C03297=1012.190,127.590,372.422,-38.235,82.167,-37.677
C03298=1012.191,127.196,372.461,-38.212,82.154,-37.653
C03299=1012.192,126.801,372.501,-38.192,82.142,-37.634
C03300=1012.193,126.407,372.540,-38.172,82.129,-37.614
C03301=1012.195,126.013,372.579,-38.150,82.117,-37.591
C03302=1012.196,125.619,372.619,-38.125,82.102,-37.566
C03303=1012.198,125.225,372.658,-38.104,82.088,-37.545
C03304=1012.199,124.830,372.698,-38.081,82.075,-37.522
C03305=1012.201,124.436,372.737,-38.059,82.062,-37.499
C03306=1012.202,124.041,372.776,-38.040,82.049,-37.481
C03307=1012.204,123.647,372.815,-38.017,82.037,-37.457
C03308=1012.205,123.254,372.854,-37.998,82.025,-37.438
C03309=1012.206,122.859,372.893,-37.978,82.013,-37.419
C03310=1012.208,122.465,372.932,-37.957,81.999,-37.398
C03311=1012.209,122.070,372.972,-37.935,81.986,-37.376
C03312=1012.210,121.676,373.012,-37.915,81.972,-37.355
C03313=1012.211,121.282,373.050,-37.893,81.959,-37.333
C03314=1012.213,120.888,373.089,-37.874,81.947,-37.314
C03315=1012.215,120.493,373.128,-37.855,81.935,-37.296
C03316=1012.216,120.099,373.167,-37.836,81.922,-37.277
C03317=1012.217,119.706,373.207,-37.817,81.911,-37.257
C03318=1012.219,119.311,373.246,-37.795,81.898,-37.235
C03319=1012.220,118.917,373.285,-37.775,81.884,-37.215
C03320=1012.222,118.523,373.324,-37.753,81.871,-37.193
C03321=1012.223,118.129,373.362,-37.736,81.858,-37.177
C03322=1012.225,117.734,373.401,-37.718,81.846,-37.159
C03323=1012.226,117.340,373.440,-37.698,81.835,-37.138
C03324=1012.227,116.945,373.479,-37.680,81.822,-37.120
C03325=1012.228,116.552,373.519,-37.662,81.810,-37.102
C03326=1012.230,116.157,373.558,-37.643,81.799,-37.083
C03327=1012.231,115.763,373.597,-37.623,81.785,-37.063
C03328=1012.232,115.369,373.636,-37.605,81.772,-37.045
C03329=1012.234,114.974,373.675,-37.584,81.759,-37.024
C03330=1012.235,114.580,373.713,-37.567,81.746,-37.009
C03331=1012.237,114.186,373.752,-37.549,81.735,-36.989
C03332=1012.238,113.792,373.791,-37.534,81.723,-36.975
C03333=1012.239,113.398,373.830,-37.515,81.712,-36.955
C03334=1012.241,113.003,373.869,-37.500,81.700,-36.941
C03335=1012.242,112.609,373.908,-37.480,81.687,-36.921
C03336=1012.244,112.215,373.947,-37.463,81.674,-36.905
C03337=1012.244,111.821,373.985,-37.443,81.661,-36.885
C03338=1012.246,111.427,374.024,-37.425,81.649,-36.867
C03339=1012.247,111.033,374.063,-37.410,81.638,-36.852
C03340=1012.249,110.638,374.101,-37.392,81.626,-36.835
C03341=1012.250,110.244,374.140,-37.377,81.615,-36.819
C03342=1012.252,109.849,374.179,-37.362,81.603,-36.805
C03343=1012.253,109.456,374.217,-37.345,81.591,-36.788
C03344=1012.255,109.062,374.256,-37.325,81.578,-36.768
C03345=1012.256,108.668,374.294,-37.308,81.566,-36.751
C03346=1012.258,108.273,374.333,-37.291,81.553,-36.735
C03347=1012.259,107.879,374.371,-37.277,81.542,-36.721
C03348=1012.260,107.484,374.410,-37.259,81.530,-36.703
C03349=1012.261,107.090,374.449,-37.245,81.518,-36.689
C03350=1012.263,106.696,374.488,-37.233,81.508,-36.678
C03351=1012.264,106.302,374.526,-37.215,81.497,-36.659
C03352=1012.266,105.907,374.565,-37.199,81.484,-36.645
C03353=1012.267,105.513,374.603,-37.182,81.471,-36.628
C03354=1012.268,105.119,374.642,-37.166,81.459,-36.612
C03355=1012.270,104.724,374.681,-37.148,81.448,-36.594
C03356=1012.271,104.330,374.719,-37.134,81.436,-36.581
C03357=1012.273,103.935,374.758,-37.120,81.425,-36.566
C03358=1012.273,103.541,374.796,-37.107,81.415,-36.554
C03359=1012.275,103.147,374.834,-37.093,81.404,-36.540
C03360=1012.276,102.752,374.873,-37.077,81.391,-36.525
C03361=1012.277,102.358,374.911,-37.061,81.379,-36.509
C03362=1012.279,101.964,374.949,-37.044,81.367,-36.491
C03363=1012.280,101.569,374.988,-37.030,81.356,-36.479
C03364=1012.281,101.175,375.026,-37.017,81.344,-36.466
C03365=1012.282,100.781,375.065,-37.002,81.333,-36.452
C03366=1012.284,100.386,375.103,-36.988,81.322,-36.437
C03367=1012.285,99.992,375.141,-36.976,81.312,-36.426
C03368=1012.286,99.598,375.180,-36.960,81.300,-36.410
C03369=1012.288,99.203,375.218,-36.947,81.288,-36.398
C03370=1012.290,98.808,375.256,-36.930,81.277,-36.380
C03371=1012.290,98.414,375.295,-36.916,81.265,-36.368
C03372=1012.292,98.019,375.332,-36.902,81.254,-36.354
C03373=1012.293,97.625,375.371,-36.889,81.242,-36.342
C03374=1012.295,97.230,375.409,-36.877,81.232,-36.331
C03375=1012.296,96.836,375.448,-36.866,81.222,-36.320
C03376=1012.297,96.442,375.485,-36.852,81.211,-36.306
C03377=1012.299,96.047,375.524,-36.836,81.199,-36.290
C03378=1012.300,95.653,375.562,-36.823,81.187,-36.278
C03379=1012.301,95.258,375.600,-36.807,81.176,-36.261
C03380=1012.302,94.863,375.638,-36.796,81.165,-36.252
C03381=1012.303,94.469,375.676,-36.782,81.154,-36.239
C03382=1012.305,94.074,375.715,-36.771,81.144,-36.228
C03383=1012.306,93.680,375.752,-36.760,81.134,-36.217
C03384=1012.307,93.286,375.791,-36.747,81.125,-36.205
C03385=1012.309,92.891,375.829,-36.735,81.113,-36.193
C03386=1012.310,92.496,375.867,-36.721,81.102,-36.179
C03387=1012.312,92.101,375.905,-36.708,81.090,-36.168
C03388=1012.313,91.707,375.943,-36.695,81.080,-36.154
C03389=1012.314,91.312,375.980,-36.682,81.068,-36.142
C03390=1012.315,90.910,376.019,-36.668,81.057,-36.129
C03391=1012.316,90.664,376.042,-36.663,81.051,-36.124
C03392=1012.317,90.384,376.070,-36.654,81.044,-36.116
C03393=1012.317,90.109,376.096,-36.646,81.037,-36.108
C03394=1012.318,89.874,376.119,-36.639,81.031,-36.101
C03395=1012.320,89.479,376.157,-36.628,81.021,-36.091
C03396=1012.321,89.094,376.194,-36.615,81.010,-36.077
C03397=1012.322,88.716,376.230,-36.604,81.000,-36.067
C03398=1012.324,88.341,376.266,-36.593,80.990,-36.057
C03399=1012.324,87.964,376.302,-36.582,80.980,-36.047
C03400=1012.326,87.579,376.340,-36.571,80.970,-36.037
C03401=1012.327,87.184,376.378,-36.561,80.960,-36.027
C03402=1012.328,86.786,376.416,-36.547,80.949,-36.013
C03403=1012.329,86.385,376.454,-36.536,80.939,-36.003
C03404=1012.331,85.983,376.492,-36.524,80.927,-35.992
C03405=1012.332,85.580,376.530,-36.514,80.917,-35.982
C03406=1012.334,85.176,376.569,-36.503,80.907,-35.972
C03407=1012.335,84.770,376.608,-36.490,80.896,-35.959
C03408=1012.335,84.363,376.647,-36.479,80.886,-35.949
C03409=1012.337,83.954,376.686,-36.467,80.874,-35.938
C03410=1012.338,83.545,376.725,-36.457,80.864,-35.928
C03411=1012.340,83.134,376.764,-36.446,80.854,-35.918
C03412=1012.340,82.722,376.804,-36.433,80.843,-35.905
C03413=1012.342,82.309,376.843,-36.423,80.833,-35.896
C03414=1012.343,81.896,376.883,-36.413,80.822,-35.888
C03415=1012.344,81.481,376.922,-36.400,80.811,-35.875
C03416=1012.346,81.087,376.960,-36.390,80.801,-35.865
C03417=1012.346,80.723,376.994,-36.381,80.792,-35.857
C03418=1012.348,80.340,377.030,-36.370,80.782,-35.847
C03419=1012.349,79.928,377.069,-36.360,80.772,-35.837
C03420=1012.351,79.520,377.108,-36.350,80.762,-35.828
C03421=1012.352,79.117,377.147,-36.339,80.751,-35.818
C03422=1012.352,78.723,377.184,-36.329,80.741,-35.809
C03423=1012.354,78.334,377.221,-36.319,80.731,-35.799
C03424=1012.355,77.950,377.258,-36.310,80.722,-35.791
C03425=1012.356,77.569,377.293,-36.300,80.712,-35.781
C03426=1012.357,77.187,377.330,-36.291,80.704,-35.773
C03427=1012.358,76.800,377.367,-36.281,80.694,-35.763
C03428=1012.359,76.406,377.403,-36.273,80.684,-35.757
C03429=1012.361,76.005,377.442,-36.263,80.674,-35.747
C03430=1012.362,75.595,377.480,-36.253,80.664,-35.738
C03431=1012.363,75.181,377.520,-36.242,80.654,-35.729
C03432=1012.364,74.972,377.539,-36.239,80.649,-35.726
C03433=1012.364,74.757,377.559,-36.232,80.643,-35.719
C03434=1012.365,74.530,377.581,-36.226,80.638,-35.713
C03435=1012.365,74.302,377.602,-36.220,80.633,-35.707
C03436=1012.366,74.083,377.623,-36.216,80.628,-35.704
C03437=1012.367,73.669,377.662,-36.206,80.618,-35.695
C03438=1012.368,73.257,377.701,-36.196,80.607,-35.685
C03439=1012.370,72.847,377.740,-36.186,80.597,-35.676
C03440=1012.371,72.439,377.778,-36.179,80.588,-35.670
C03441=1012.372,72.032,377.816,-36.169,80.578,-35.661
C03442=1012.373,71.628,377.854,-36.160,80.569,-35.653
C03443=1012.375,71.223,377.893,-36.150,80.559,-35.644
C03444=1012.375,70.818,377.931,-36.140,80.549,-35.634
C03445=1012.377,70.414,377.969,-36.133,80.539,-35.628
C03446=1012.378,70.010,378.006,-36.124,80.531,-35.620
C03447=1012.378,69.606,378.045,-36.115,80.520,-35.611
C03448=1012.379,69.198,378.083,-36.107,80.511,-35.605
C03449=1012.381,68.782,378.122,-36.096,80.502,-35.594
C03450=1012.382,68.364,378.161,-36.089,80.492,-35.588
C03451=1012.383,67.953,378.199,-36.079,80.482,-35.579
C03452=1012.384,67.552,378.237,-36.071,80.473,-35.571
C03453=1012.385,67.153,378.275,-36.063,80.464,-35.565
C03454=1012.386,66.756,378.311,-36.056,80.454,-35.559
C03455=1012.387,66.393,378.346,-36.047,80.447,-35.550
C03456=1012.388,66.065,378.376,-36.041,80.439,-35.545
C03457=1012.390,65.672,378.412,-36.032,80.430,-35.537
C03458=1012.390,65.464,378.433,-36.029,80.425,-35.534
C03459=1012.391,65.249,378.452,-36.025,80.421,-35.531
C03460=1012.391,65.030,378.473,-36.019,80.415,-35.525
C03461=1012.391,64.808,378.493,-36.015,80.410,-35.522
C03462=1012.392,64.582,378.515,-36.009,80.405,-35.516
C03463=1012.393,64.355,378.536,-36.006,80.400,-35.513
C03464=1012.393,64.136,378.556,-36.002,80.395,-35.510
C03465=1012.395,63.730,378.593,-35.955,80.352,-35.464
C03466=1012.395,63.519,378.609,-35.868,80.276,-35.376
C03467=1012.397,63.284,378.627,-35.774,80.189,-35.282
C03468=1012.398,63.036,378.646,-35.677,80.098,-35.185
C03469=1012.400,62.794,378.664,-35.583,80.009,-35.091
C03470=1012.401,62.574,378.681,-35.501,79.929,-35.008
C03471=1012.402,62.291,378.703,-35.396,79.825,-34.903
C03472=1012.404,61.892,378.733,-35.253,79.680,-34.760
C03473=1012.406,61.497,378.763,-35.115,79.536,-34.622
C03474=1012.408,61.100,378.794,-34.981,79.393,-34.488
C03475=1012.409,60.704,378.824,-34.851,79.248,-34.359
C03476=1012.412,60.307,378.854,-34.727,79.105,-34.236
C03477=1012.413,59.912,378.885,-34.605,78.962,-34.114
C03478=1012.415,59.516,378.916,-34.487,78.819,-33.997
C03479=1012.418,59.120,378.945,-34.374,78.677,-33.885
C03480=1012.420,58.724,378.976,-34.264,78.535,-33.777
C03481=1012.422,58.327,379.006,-34.156,78.393,-33.670
C03482=1012.423,57.932,379.036,-34.051,78.251,-33.567
C03483=1012.426,57.535,379.067,-33.951,78.110,-33.468
C03484=1012.428,57.140,379.097,-33.853,77.969,-33.372
C03485=1012.430,56.743,379.127,-33.756,77.828,-33.278
C03486=1012.432,56.347,379.158,-33.663,77.688,-33.186
C03487=1012.434,55.950,379.188,-33.573,77.548,-33.098
C03488=1012.436,55.555,379.218,-33.485,77.407,-33.013
C03489=1012.438,55.159,379.249,-33.400,77.267,-32.931
C03490=1012.441,54.763,379.279,-33.317,77.128,-32.851
C03491=1012.442,54.367,379.310,-33.236,76.990,-32.773
C03492=1012.445,53.971,379.340,-33.157,76.851,-32.697
C03493=1012.447,53.575,379.371,-33.081,76.713,-32.624
C03494=1012.449,53.179,379.400,-33.007,76.575,-32.554
C03495=1012.452,52.783,379.431,-32.934,76.437,-32.485
C03496=1012.454,52.387,379.461,-32.862,76.300,-32.417
C03497=1012.455,51.991,379.491,-32.793,76.163,-32.352
C03498=1012.458,51.596,379.522,-32.725,76.027,-32.288
C03499=1012.460,51.199,379.552,-32.660,75.890,-32.227
C03500=1012.462,50.804,379.582,-32.597,75.754,-32.168
C03501=1012.465,50.407,379.613,-32.534,75.619,-32.109
C03502=1012.467,50.011,379.644,-32.473,75.483,-32.054
C03503=1012.469,49.616,379.674,-32.412,75.348,-31.998
C03504=1012.471,49.219,379.704,-32.355,75.214,-31.945
C03505=1012.474,48.824,379.734,-32.297,75.080,-31.892
C03506=1012.475,48.428,379.765,-32.243,74.946,-31.844
C03507=1012.478,48.032,379.795,-32.189,74.813,-31.795
C03508=1012.480,47.636,379.826,-32.136,74.680,-31.747
C03509=1012.481,47.241,379.856,-32.084,74.547,-31.701
C03510=1012.484,46.845,379.886,-32.034,74.415,-31.658
C03511=1012.487,46.449,379.916,-31.985,74.283,-31.614
C03512=1012.488,46.054,379.947,-31.936,74.151,-31.571
C03513=1012.491,45.658,379.977,-31.889,74.020,-31.531
C03514=1012.493,45.262,380.007,-31.843,73.890,-31.490
C03515=1012.495,44.867,380.038,-31.798,73.759,-31.452
C03516=1012.498,44.470,380.068,-31.753,73.628,-31.414
C03517=1012.500,44.075,380.098,-31.710,73.498,-31.378
C03518=1012.502,43.679,380.129,-31.668,73.370,-31.342
C03519=1012.504,43.283,380.159,-31.627,73.240,-31.308
C03520=1012.507,42.888,380.189,-31.586,73.112,-31.275
C03521=1012.509,42.492,380.220,-31.546,72.984,-31.242
C03522=1012.511,42.096,380.250,-31.508,72.856,-31.212
C03523=1012.513,41.701,380.280,-31.470,72.729,-31.181
C03524=1012.515,41.305,380.311,-31.432,72.602,-31.150
C03525=1012.518,40.909,380.341,-31.395,72.476,-31.121
C03526=1012.520,40.514,380.371,-31.360,72.349,-31.094
C03527=1012.522,40.118,380.402,-31.326,72.224,-31.069
C03528=1012.524,39.723,380.432,-31.291,72.098,-31.041
C03529=1012.527,39.328,380.463,-31.258,71.973,-31.016
C03530=1012.530,38.932,380.493,-31.225,71.850,-30.991
C03531=1012.531,38.536,380.523,-31.192,71.725,-30.967
C03532=1012.534,38.141,380.554,-31.160,71.602,-30.944
C03533=1012.536,37.746,380.584,-31.130,71.480,-30.922
C03534=1012.539,37.351,380.614,-31.100,71.357,-30.902
C03535=1012.541,36.954,380.645,-31.070,71.235,-30.880
C03536=1012.543,36.559,380.675,-31.041,71.114,-30.860
C03537=1012.545,36.164,380.706,-31.012,70.993,-30.840
C03538=1012.548,35.768,380.735,-30.984,70.872,-30.822
C03539=1012.550,35.372,380.766,-30.957,70.752,-30.803
C03540=1012.552,34.977,380.797,-30.929,70.632,-30.785
C03541=1012.554,34.582,380.827,-30.903,70.513,-30.768
C03542=1012.557,34.187,380.857,-30.877,70.394,-30.752
C03543=1012.559,33.792,380.887,-30.851,70.276,-30.736
C03544=1012.561,33.396,380.918,-30.826,70.158,-30.721
C03545=1012.564,33.000,380.949,-30.802,70.041,-30.706
C03546=1012.565,32.605,380.979,-30.777,69.924,-30.691
C03547=1012.568,32.210,381.009,-30.754,69.807,-30.679
C03548=1012.570,31.815,381.039,-30.730,69.691,-30.665
C03549=1012.573,31.420,381.070,-30.707,69.576,-30.651
C03550=1012.574,31.024,381.100,-30.684,69.461,-30.640
C03551=1012.577,30.629,381.131,-30.663,69.347,-30.628
C03552=1012.579,30.233,381.161,-30.640,69.233,-30.616
C03553=1012.581,29.838,381.191,-30.619,69.119,-30.606
C03554=1012.584,29.443,381.222,-30.599,69.006,-30.597
C03555=1012.586,29.048,381.252,-30.578,68.893,-30.586
C03556=1012.589,28.652,381.283,-30.558,68.782,-30.578
C03557=1012.591,28.259,381.313,-30.537,68.671,-30.567
C03558=1012.593,27.865,381.343,-30.518,68.561,-30.559
C03559=1012.595,27.473,381.373,-30.499,68.451,-30.551
C03560=1012.597,27.079,381.404,-30.480,68.341,-30.544
C03561=1012.599,26.684,381.434,-30.461,68.232,-30.535
C03562=1012.601,26.288,381.465,-30.443,68.122,-30.529
C03563=1012.604,25.890,381.495,-30.426,68.013,-30.523
C03564=1012.606,25.493,381.526,-30.408,67.905,-30.517
C03565=1012.608,25.096,381.556,-30.390,67.796,-30.511
C03566=1012.611,24.701,381.587,-30.373,67.689,-30.504
C03567=1012.613,24.305,381.618,-30.356,67.583,-30.500
C03568=1012.615,23.926,381.646,-30.340,67.481,-30.496
C03569=1012.617,23.585,381.673,-30.326,67.390,-30.491
C03570=1012.619,23.169,381.705,-30.309,67.280,-30.486
C03571=1012.621,22.805,381.733,-30.294,67.184,-30.483
C03572=1012.623,22.529,381.754,-30.283,67.111,-30.480
C03573=1012.624,22.198,381.779,-30.270,67.024,-30.476
C03574=1012.626,21.869,381.805,-30.258,66.938,-30.475
C03575=1012.628,21.481,381.835,-30.243,66.837,-30.472
C03576=1012.629,21.253,381.852,-30.234,66.778,-30.470
C03577=1012.631,21.005,381.872,-30.225,66.715,-30.468
C03578=1012.632,20.744,381.891,-30.215,66.647,-30.465
C03579=1012.634,20.476,381.912,-30.205,66.578,-30.464
C03580=1012.635,20.206,381.933,-30.196,66.509,-30.463
C03581=1012.636,19.946,381.953,-30.187,66.443,-30.463
C03582=1012.638,19.704,381.972,-30.178,66.382,-30.461
C03583=1012.640,19.483,381.989,-30.170,66.326,-30.460
C03584=1012.640,19.279,382.004,-30.163,66.274,-30.460
C03585=1012.643,18.877,382.035,-30.149,66.173,-30.459
C03586=1012.644,18.478,382.066,-30.136,66.072,-30.458
C03587=1012.647,18.086,382.096,-30.123,65.976,-30.457
C03588=1012.649,17.696,382.127,-30.110,65.879,-30.456
C03589=1012.651,17.308,382.157,-30.097,65.784,-30.455
C03590=1012.653,16.922,382.186,-30.085,65.690,-30.456
C03591=1012.655,16.538,382.215,-30.073,65.596,-30.456
C03592=1012.657,16.155,382.245,-30.061,65.503,-30.456
C03593=1012.659,15.774,382.274,-30.049,65.412,-30.456
C03594=1012.660,15.393,382.304,-30.038,65.320,-30.458
C03595=1012.663,15.013,382.333,-30.027,65.230,-30.460
C03596=1012.665,14.633,382.362,-30.015,65.141,-30.460
C03597=1012.667,14.253,382.392,-30.004,65.050,-30.461
C03598=1012.668,13.871,382.421,-29.993,64.962,-30.463
C03599=1012.671,13.490,382.451,-29.982,64.873,-30.464
C03600=1012.673,13.108,382.481,-29.972,64.784,-30.466
C03601=1012.674,12.724,382.510,-29.962,64.696,-30.469
C03602=1012.676,12.340,382.539,-29.951,64.609,-30.469
C03603=1012.678,11.957,382.569,-29.941,64.522,-30.472
C03604=1012.680,11.585,382.598,-29.931,64.438,-30.475
C03605=1012.682,11.222,382.626,-29.921,64.355,-30.478
C03606=1012.684,10.856,382.654,-29.912,64.275,-30.480
C03607=1012.686,10.483,382.683,-29.903,64.192,-30.483
C03608=1012.688,10.105,382.712,-29.893,64.108,-30.486
C03609=1012.690,9.729,382.741,-29.884,64.026,-30.490
C03610=1012.692,9.354,382.770,-29.875,63.944,-30.492
C03611=1012.693,8.981,382.799,-29.866,63.864,-30.495
C03612=1012.695,8.607,382.828,-29.857,63.784,-30.500
C03613=1012.697,8.233,382.857,-29.849,63.703,-30.503
C03614=1012.699,7.857,382.886,-29.840,63.624,-30.507
C03615=1012.701,7.479,382.915,-29.831,63.544,-30.511
C03616=1012.702,7.097,382.944,-29.823,63.464,-30.515
C03617=1012.704,6.712,382.974,-29.814,63.385,-30.518
C03618=1012.706,6.321,383.004,-29.806,63.303,-30.524
C03619=1012.708,5.928,383.034,-29.797,63.222,-30.528
C03620=1012.710,5.535,383.065,-29.789,63.143,-30.532
C03621=1012.711,5.144,383.095,-29.781,63.064,-30.538
C03622=1012.713,4.756,383.125,-29.773,62.987,-30.542
C03623=1012.715,4.367,383.155,-29.765,62.908,-30.547
C03624=1012.717,3.976,383.185,-29.757,62.832,-30.551
C03625=1012.719,3.603,383.214,-29.750,62.758,-30.557
C03626=1012.720,3.259,383.241,-29.743,62.691,-30.562
C03627=1012.721,2.935,383.266,-29.737,62.629,-30.566
C03628=1012.723,2.612,383.291,-29.731,62.567,-30.571
C03629=1012.725,2.270,383.317,-29.724,62.502,-30.575
C03630=1012.726,1.899,383.346,-29.717,62.431,-30.580
